	MoveL Offs(p0,126.52000000000001,464.52479999999997, 0), v100, z5, tool0;
	MoveL Offs(p0,127.525,466.325, 0), v100, z5, tool0;
	MoveL Offs(p0,128.584,468.0831999999999, 0), v100, z5, tool0;
	MoveL Offs(p0,129.679,469.7646, 0), v100, z5, tool0;
	MoveL Offs(p0,130.792,471.3344000000001, 0), v100, z5, tool0;
	MoveL Offs(p0,131.90500000000003,472.75780000000003, 0), v100, z5, tool0;
	MoveL Offs(p0,133.0,474.0, 0), v100, z5, tool0;
	MoveL Offs(p0,137.77200000000002,479.7586, 0), v100, z5, tool0;
	MoveL Offs(p0,142.54400000000004,486.68480000000017, 0), v100, z5, tool0;
	MoveL Offs(p0,147.22,494.55420000000004, 0), v100, z5, tool0;
	MoveL Offs(p0,151.704,503.14240000000007, 0), v100, z5, tool0;
	MoveL Offs(p0,155.9,512.225, 0), v100, z5, tool0;
	MoveL Offs(p0,159.712,521.5776, 0), v100, z5, tool0;
	MoveL Offs(p0,163.044,530.9757999999999, 0), v100, z5, tool0;
	MoveL Offs(p0,165.8,540.1952, 0), v100, z5, tool0;
	MoveL Offs(p0,167.884,549.0114000000001, 0), v100, z5, tool0;
	MoveL Offs(p0,169.2,557.2, 0), v100, z5, tool0;
	MoveL Offs(p0,169.67680000000001,561.0432000000002, 0), v100, z5, tool0;
	MoveL Offs(p0,169.9092,562.9168000000001, 0), v100, z5, tool0;
	MoveL Offs(p0,170.1344,564.7136, 0), v100, z5, tool0;
	MoveL Offs(p0,170.35,566.4, 0), v100, z5, tool0;
	MoveL Offs(p0,170.5536,567.9424, 0), v100, z5, tool0;
	MoveL Offs(p0,170.7428,569.3072, 0), v100, z5, tool0;
	MoveL Offs(p0,170.9152,570.4608000000001, 0), v100, z5, tool0;
	MoveL Offs(p0,171.06840000000003,571.3696, 0), v100, z5, tool0;
	MoveL Offs(p0,171.2,572.0, 0), v100, z5, tool0;
	MoveL Offs(p0,171.4976,574.6176, 0), v100, z5, tool0;
	MoveL Offs(p0,171.575,575.425, 0), v100, z5, tool0;
	MoveL Offs(p0,171.6464,576.2624, 0), v100, z5, tool0;
	MoveL Offs(p0,171.7082,577.1142, 0), v100, z5, tool0;
	MoveL Offs(p0,171.75680000000003,577.9648, 0), v100, z5, tool0;
	MoveL Offs(p0,171.78860000000003,578.7986000000001, 0), v100, z5, tool0;
	MoveL Offs(p0,171.8,579.6, 0), v100, z5, tool0;
	MoveL Offs(p0,172.0772,581.6088, 0), v100, z5, tool0;
	MoveL Offs(p0,172.20640000000003,582.1856, 0), v100, z5, tool0;
	MoveL Offs(p0,172.35,582.7, 0), v100, z5, tool0;
	MoveL Offs(p0,172.50560000000002,583.1424, 0), v100, z5, tool0;
	MoveL Offs(p0,172.6708,583.5032, 0), v100, z5, tool0;
	MoveL Offs(p0,172.84320000000002,583.7728000000001, 0), v100, z5, tool0;
	MoveL Offs(p0,173.02040000000002,583.9416, 0), v100, z5, tool0;
	MoveL Offs(p0,173.2,584.0, 0), v100, z5, tool0;
	MoveL Offs(p0,173.70940000000002,581.9156, 0), v100, z5, tool0;
	MoveL Offs(p0,173.7888,580.4032, 0), v100, z5, tool0;
	MoveL Offs(p0,173.825,578.55, 0), v100, z5, tool0;
	MoveL Offs(p0,173.8192,576.3968, 0), v100, z5, tool0;
	MoveL Offs(p0,173.7726,573.9844, 0), v100, z5, tool0;
	MoveL Offs(p0,173.6864,571.3536, 0), v100, z5, tool0;
	MoveL Offs(p0,173.5618,568.5452, 0), v100, z5, tool0;
	MoveL Offs(p0,173.4,565.6, 0), v100, z5, tool0;
	MoveL Offs(p0,173.4,565.6, 0), v100, z5, tool0;
	MoveJ Offs(p0,300.6,571.2, 10), v100, z1, tool0;
	MoveL Offs(p0,301.2482,569.1882, 0), v100, z5, tool0;
	MoveL Offs(p0,301.75360000000006,567.4416000000002, 0), v100, z5, tool0;
	MoveL Offs(p0,302.1174,565.9134000000001, 0), v100, z5, tool0;
	MoveL Offs(p0,302.34080000000006,564.5568000000001, 0), v100, z5, tool0;
	MoveL Offs(p0,302.425,563.325, 0), v100, z5, tool0;
	MoveL Offs(p0,302.37119999999993,562.1712, 0), v100, z5, tool0;
	MoveL Offs(p0,302.18059999999997,561.0486, 0), v100, z5, tool0;
	MoveL Offs(p0,301.85440000000006,559.9104, 0), v100, z5, tool0;
	MoveL Offs(p0,301.3938,558.7098, 0), v100, z5, tool0;
	MoveL Offs(p0,300.8,557.4, 0), v100, z5, tool0;
	MoveL Offs(p0,298.2224,550.942, 0), v100, z5, tool0;
	MoveL Offs(p0,296.3552000000001,542.8880000000001, 0), v100, z5, tool0;
	MoveL Offs(p0,295.1768,533.658, 0), v100, z5, tool0;
	MoveL Offs(p0,294.66560000000004,523.672, 0), v100, z5, tool0;
	MoveL Offs(p0,294.8,513.35, 0), v100, z5, tool0;
	MoveL Offs(p0,295.5584,503.11199999999997, 0), v100, z5, tool0;
	MoveL Offs(p0,296.9192,493.37800000000004, 0), v100, z5, tool0;
	MoveL Offs(p0,298.86080000000004,484.56800000000004, 0), v100, z5, tool0;
	MoveL Offs(p0,301.36160000000007,477.10200000000003, 0), v100, z5, tool0;
	MoveL Offs(p0,304.4,471.4, 0), v100, z5, tool0;
	MoveL Offs(p0,306.18019999999996,468.8188, 0), v100, z5, tool0;
	MoveL Offs(p0,306.66240000000005,468.0496, 0), v100, z5, tool0;
	MoveL Offs(p0,307.075,467.35, 0), v100, z5, tool0;
	MoveL Offs(p0,307.4096,466.7344, 0), v100, z5, tool0;
	MoveL Offs(p0,307.6578,466.21719999999993, 0), v100, z5, tool0;
	MoveL Offs(p0,307.8112,465.81280000000004, 0), v100, z5, tool0;
	MoveL Offs(p0,307.8614,465.53560000000004, 0), v100, z5, tool0;
	MoveL Offs(p0,307.8,465.4, 0), v100, z5, tool0;
	MoveL Offs(p0,305.02880000000005,464.32320000000016, 0), v100, z5, tool0;
	MoveL Offs(p0,302.53319999999997,463.44879999999995, 0), v100, z5, tool0;
	MoveL Offs(p0,299.5984,462.44960000000003, 0), v100, z5, tool0;
	MoveL Offs(p0,296.45,461.4, 0), v100, z5, tool0;
	MoveL Offs(p0,293.3136,460.3744, 0), v100, z5, tool0;
	MoveL Offs(p0,290.4148,459.44719999999995, 0), v100, z5, tool0;
	MoveL Offs(p0,287.97920000000005,458.6928, 0), v100, z5, tool0;
	MoveL Offs(p0,286.2324,458.1856000000001, 0), v100, z5, tool0;
	MoveL Offs(p0,285.4,458.0, 0), v100, z5, tool0;
	MoveL Offs(p0,283.55499999999995,460.51099999999997, 0), v100, z5, tool0;
	MoveL Offs(p0,282.80800000000005,462.32000000000005, 0), v100, z5, tool0;
	MoveL Offs(p0,282.025,464.525, 0), v100, z5, tool0;
	MoveL Offs(p0,281.224,467.072, 0), v100, z5, tool0;
	MoveL Offs(p0,280.423,469.90700000000004, 0), v100, z5, tool0;
	MoveL Offs(p0,279.64000000000004,472.976, 0), v100, z5, tool0;
	MoveL Offs(p0,278.89300000000003,476.225, 0), v100, z5, tool0;
	MoveL Offs(p0,278.2,479.6, 0), v100, z5, tool0;
	MoveL Offs(p0,276.93420000000003,487.9902000000001, 0), v100, z5, tool0;
	MoveL Offs(p0,276.2336000000001,497.66560000000015, 0), v100, z5, tool0;
	MoveL Offs(p0,276.0634,508.2434, 0), v100, z5, tool0;
	MoveL Offs(p0,276.38880000000006,519.3408000000001, 0), v100, z5, tool0;
	MoveL Offs(p0,277.175,530.575, 0), v100, z5, tool0;
	MoveL Offs(p0,278.3872,541.5631999999999, 0), v100, z5, tool0;
	MoveL Offs(p0,279.9906,551.9226, 0), v100, z5, tool0;
	MoveL Offs(p0,281.9504,561.2704, 0), v100, z5, tool0;
	MoveL Offs(p0,284.2318,569.2238, 0), v100, z5, tool0;
	MoveL Offs(p0,286.8,575.4, 0), v100, z5, tool0;
	MoveL Offs(p0,288.153,577.6692, 0), v100, z5, tool0;
	MoveL Offs(p0,289.56000000000006,579.3216000000002, 0), v100, z5, tool0;
	MoveL Offs(p0,291.003,580.3644, 0), v100, z5, tool0;
	MoveL Offs(p0,292.46400000000006,580.8048, 0), v100, z5, tool0;
	MoveL Offs(p0,293.925,580.65, 0), v100, z5, tool0;
	MoveL Offs(p0,295.368,579.9071999999999, 0), v100, z5, tool0;
	MoveL Offs(p0,296.775,578.5836, 0), v100, z5, tool0;
	MoveL Offs(p0,298.12800000000004,576.6864, 0), v100, z5, tool0;
	MoveL Offs(p0,299.409,574.2228000000001, 0), v100, z5, tool0;
	MoveL Offs(p0,300.6,571.2, 0), v100, z5, tool0;
	MoveL Offs(p0,300.6,571.2, 0), v100, z5, tool0;
	MoveJ Offs(p0,313.0,572.2, 10), v100, z1, tool0;
	MoveL Offs(p0,312.6486000000001,570.0876000000001, 0), v100, z5, tool0;
	MoveL Offs(p0,312.56480000000005,568.0448000000001, 0), v100, z5, tool0;
	MoveL Offs(p0,312.76419999999996,566.0332, 0), v100, z5, tool0;
	MoveL Offs(p0,313.2624,564.0143999999999, 0), v100, z5, tool0;
	MoveL Offs(p0,314.075,561.95, 0), v100, z5, tool0;
	MoveL Offs(p0,315.2176,559.8016, 0), v100, z5, tool0;
	MoveL Offs(p0,316.7058,557.5308, 0), v100, z5, tool0;
	MoveL Offs(p0,318.55520000000007,555.0992, 0), v100, z5, tool0;
	MoveL Offs(p0,320.7814,552.4684, 0), v100, z5, tool0;
	MoveL Offs(p0,323.4,549.6, 0), v100, z5, tool0;
	MoveL Offs(p0,325.2538,547.5742000000001, 0), v100, z5, tool0;
	MoveL Offs(p0,326.7344000000001,545.7056000000002, 0), v100, z5, tool0;
	MoveL Offs(p0,327.84059999999994,544.0074000000001, 0), v100, z5, tool0;
	MoveL Offs(p0,328.5712,542.4928, 0), v100, z5, tool0;
	MoveL Offs(p0,328.925,541.175, 0), v100, z5, tool0;
	MoveL Offs(p0,328.9008,540.0672, 0), v100, z5, tool0;
	MoveL Offs(p0,328.4974,539.1826, 0), v100, z5, tool0;
	MoveL Offs(p0,327.71360000000004,538.5344000000001, 0), v100, z5, tool0;
	MoveL Offs(p0,326.54820000000007,538.1358, 0), v100, z5, tool0;
	MoveL Offs(p0,325.0,538.0, 0), v100, z5, tool0;
	MoveL Offs(p0,321.8720000000001,541.2496000000001, 0), v100, z5, tool0;
	MoveL Offs(p0,319.573,544.8093999999999, 0), v100, z5, tool0;
	MoveL Offs(p0,317.016,549.2128, 0), v100, z5, tool0;
	MoveL Offs(p0,314.375,554.125, 0), v100, z5, tool0;
	MoveL Offs(p0,311.824,559.2112, 0), v100, z5, tool0;
	MoveL Offs(p0,309.537,564.1366, 0), v100, z5, tool0;
	MoveL Offs(p0,307.688,568.5664, 0), v100, z5, tool0;
	MoveL Offs(p0,306.451,572.1658, 0), v100, z5, tool0;
	MoveL Offs(p0,306.0,574.6, 0), v100, z5, tool0;
	MoveL Offs(p0,306.7296,576.7472, 0), v100, z5, tool0;
	MoveL Offs(p0,307.125,577.125, 0), v100, z5, tool0;
	MoveL Offs(p0,307.59839999999997,577.4368, 0), v100, z5, tool0;
	MoveL Offs(p0,308.1462,577.6814, 0), v100, z5, tool0;
	MoveL Offs(p0,308.76480000000004,577.8576, 0), v100, z5, tool0;
	MoveL Offs(p0,309.4506,577.9642000000001, 0), v100, z5, tool0;
	MoveL Offs(p0,310.2,578.0, 0), v100, z5, tool0;
	MoveL Offs(p0,312.6192,577.6922, 0), v100, z5, tool0;
	MoveL Offs(p0,313.0864,577.3984, 0), v100, z5, tool0;
	MoveL Offs(p0,313.4,576.975, 0), v100, z5, tool0;
	MoveL Offs(p0,313.56960000000004,576.4015999999999, 0), v100, z5, tool0;
	MoveL Offs(p0,313.60479999999995,575.6578000000001, 0), v100, z5, tool0;
	MoveL Offs(p0,313.5152,574.7232, 0), v100, z5, tool0;
	MoveL Offs(p0,313.3104,573.5774, 0), v100, z5, tool0;
	MoveL Offs(p0,313.0,572.2, 0), v100, z5, tool0;
	MoveL Offs(p0,313.0,572.2, 0), v100, z5, tool0;
	MoveJ Offs(p0,343.8,570.4, 10), v100, z1, tool0;
	MoveL Offs(p0,360.4,567.0, 0), v100, z5, tool0;
	MoveL Offs(p0,348.2,557.2, 0), v100, z5, tool0;
	MoveL Offs(p0,344.5584,554.3928000000002, 0), v100, z5, tool0;
	MoveL Offs(p0,341.5792,552.2144000000001, 0), v100, z5, tool0;
	MoveL Offs(p0,339.1208,550.6696, 0), v100, z5, tool0;
	MoveL Offs(p0,337.0416000000001,549.7632000000001, 0), v100, z5, tool0;
	MoveL Offs(p0,335.2,549.5, 0), v100, z5, tool0;
	MoveL Offs(p0,333.45439999999996,549.8848, 0), v100, z5, tool0;
	MoveL Offs(p0,331.6632,550.9224, 0), v100, z5, tool0;
	MoveL Offs(p0,329.68480000000005,552.6176, 0), v100, z5, tool0;
	MoveL Offs(p0,327.3776,554.9752000000001, 0), v100, z5, tool0;
	MoveL Offs(p0,324.6,558.0, 0), v100, z5, tool0;
	MoveL Offs(p0,322.8896000000001,560.1758000000002, 0), v100, z5, tool0;
	MoveL Offs(p0,321.59680000000014,562.3504000000001, 0), v100, z5, tool0;
	MoveL Offs(p0,320.71919999999994,564.4746, 0), v100, z5, tool0;
	MoveL Offs(p0,320.25440000000003,566.4992, 0), v100, z5, tool0;
	MoveL Offs(p0,320.2,568.375, 0), v100, z5, tool0;
	MoveL Offs(p0,320.55359999999996,570.0527999999999, 0), v100, z5, tool0;
	MoveL Offs(p0,321.3128,571.4834, 0), v100, z5, tool0;
	MoveL Offs(p0,322.47520000000003,572.6176, 0), v100, z5, tool0;
	MoveL Offs(p0,324.0384,573.4062, 0), v100, z5, tool0;
	MoveL Offs(p0,326.0,573.8, 0), v100, z5, tool0;
	MoveL Offs(p0,328.3706,573.4057999999999, 0), v100, z5, tool0;
	MoveL Offs(p0,329.87520000000006,573.1216000000001, 0), v100, z5, tool0;
	MoveL Offs(p0,331.675,572.775, 0), v100, z5, tool0;
	MoveL Offs(p0,333.73279999999994,572.3743999999999, 0), v100, z5, tool0;
	MoveL Offs(p0,336.0114,571.9282000000001, 0), v100, z5, tool0;
	MoveL Offs(p0,338.47360000000003,571.4448, 0), v100, z5, tool0;
	MoveL Offs(p0,341.0822,570.9326, 0), v100, z5, tool0;
	MoveL Offs(p0,343.8,570.4, 0), v100, z5, tool0;
	MoveL Offs(p0,343.8,570.4, 0), v100, z5, tool0;
	MoveJ Offs(p0,145.8,567.6, 10), v100, z1, tool0;
	MoveL Offs(p0,148.6,563.2, 0), v100, z5, tool0;
	MoveL Offs(p0,152.0,567.6, 0), v100, z5, tool0;
	MoveL Offs(p0,154.31040000000002,570.2736000000001, 0), v100, z5, tool0;
	MoveL Offs(p0,155.18959999999998,571.0794, 0), v100, z5, tool0;
	MoveL Offs(p0,155.9392,571.5168000000001, 0), v100, z5, tool0;
	MoveL Offs(p0,156.6,571.575, 0), v100, z5, tool0;
	MoveL Offs(p0,157.2128,571.2432000000001, 0), v100, z5, tool0;
	MoveL Offs(p0,157.8184,570.5106, 0), v100, z5, tool0;
	MoveL Offs(p0,158.4576,569.3664000000001, 0), v100, z5, tool0;
	MoveL Offs(p0,159.1712,567.7998, 0), v100, z5, tool0;
	MoveL Offs(p0,160.0,565.8, 0), v100, z5, tool0;
	MoveL Offs(p0,161.5264,563.019, 0), v100, z5, tool0;
	MoveL Offs(p0,162.06080000000003,562.3120000000001, 0), v100, z5, tool0;
	MoveL Offs(p0,162.6,561.725, 0), v100, z5, tool0;
	MoveL Offs(p0,163.13920000000002,561.2639999999999, 0), v100, z5, tool0;
	MoveL Offs(p0,163.6736,560.9350000000001, 0), v100, z5, tool0;
	MoveL Offs(p0,164.19840000000002,560.744, 0), v100, z5, tool0;
	MoveL Offs(p0,164.70880000000002,560.697, 0), v100, z5, tool0;
	MoveL Offs(p0,165.2,560.8, 0), v100, z5, tool0;
	MoveL Offs(p0,167.2,561.4, 0), v100, z5, tool0;
	MoveL Offs(p0,167.4752,561.4480000000001, 0), v100, z5, tool0;
	MoveL Offs(p0,167.69760000000002,561.472, 0), v100, z5, tool0;
	MoveL Offs(p0,167.86240000000004,561.472, 0), v100, z5, tool0;
	MoveL Offs(p0,167.96480000000003,561.4480000000001, 0), v100, z5, tool0;
	MoveL Offs(p0,168.0,561.4, 0), v100, z5, tool0;
	MoveL Offs(p0,167.65260000000004,558.7860000000001, 0), v100, z5, tool0;
	MoveL Offs(p0,166.68480000000005,554.6480000000001, 0), v100, z5, tool0;
	MoveL Offs(p0,165.20819999999998,549.322, 0), v100, z5, tool0;
	MoveL Offs(p0,163.33440000000002,543.1440000000001, 0), v100, z5, tool0;
	MoveL Offs(p0,161.175,536.45, 0), v100, z5, tool0;
	MoveL Offs(p0,158.8416,529.576, 0), v100, z5, tool0;
	MoveL Offs(p0,156.44580000000002,522.858, 0), v100, z5, tool0;
	MoveL Offs(p0,154.09920000000002,516.632, 0), v100, z5, tool0;
	MoveL Offs(p0,151.9134,511.23400000000004, 0), v100, z5, tool0;
	MoveL Offs(p0,150.0,507.0, 0), v100, z5, tool0;
	MoveL Offs(p0,147.63520000000003,502.4732, 0), v100, z5, tool0;
	MoveL Offs(p0,144.85760000000005,497.68960000000004, 0), v100, z5, tool0;
	MoveL Offs(p0,141.8424,492.8843999999999, 0), v100, z5, tool0;
	MoveL Offs(p0,138.76479999999998,488.29280000000006, 0), v100, z5, tool0;
	MoveL Offs(p0,135.8,484.15, 0), v100, z5, tool0;
	MoveL Offs(p0,133.1232,480.69120000000004, 0), v100, z5, tool0;
	MoveL Offs(p0,130.9096,478.1516, 0), v100, z5, tool0;
	MoveL Offs(p0,129.33440000000002,476.7664000000001, 0), v100, z5, tool0;
	MoveL Offs(p0,128.5728,476.77080000000007, 0), v100, z5, tool0;
	MoveL Offs(p0,128.8,478.4, 0), v100, z5, tool0;
	MoveL Offs(p0,130.18980000000002,484.4408, 0), v100, z5, tool0;
	MoveL Offs(p0,131.35040000000004,492.3824000000001, 0), v100, z5, tool0;
	MoveL Offs(p0,132.2686,501.71360000000004, 0), v100, z5, tool0;
	MoveL Offs(p0,132.93120000000002,511.9232, 0), v100, z5, tool0;
	MoveL Offs(p0,133.325,522.5, 0), v100, z5, tool0;
	MoveL Offs(p0,133.4368,532.9328, 0), v100, z5, tool0;
	MoveL Offs(p0,133.2534,542.7103999999999, 0), v100, z5, tool0;
	MoveL Offs(p0,132.7616,551.3216, 0), v100, z5, tool0;
	MoveL Offs(p0,131.94819999999999,558.2552, 0), v100, z5, tool0;
	MoveL Offs(p0,130.8,563.0, 0), v100, z5, tool0;
	MoveL Offs(p0,130.18880000000001,565.0992, 0), v100, z5, tool0;
	MoveL Offs(p0,130.225,565.375, 0), v100, z5, tool0;
	MoveL Offs(p0,130.3392,565.5487999999999, 0), v100, z5, tool0;
	MoveL Offs(p0,130.5326,565.6193999999999, 0), v100, z5, tool0;
	MoveL Offs(p0,130.8064,565.5856, 0), v100, z5, tool0;
	MoveL Offs(p0,131.16180000000003,565.4462000000001, 0), v100, z5, tool0;
	MoveL Offs(p0,131.6,565.2, 0), v100, z5, tool0;
	MoveL Offs(p0,133.925,565.4, 0), v100, z5, tool0;
	MoveL Offs(p0,134.45120000000003,565.7472, 0), v100, z5, tool0;
	MoveL Offs(p0,134.9726,566.1856, 0), v100, z5, tool0;
	MoveL Offs(p0,135.47840000000002,566.7104, 0), v100, z5, tool0;
	MoveL Offs(p0,135.9578,567.3168, 0), v100, z5, tool0;
	MoveL Offs(p0,136.4,568.0, 0), v100, z5, tool0;
	MoveL Offs(p0,138.28000000000003,570.4736000000001, 0), v100, z5, tool0;
	MoveL Offs(p0,139.19899999999998,571.2274, 0), v100, z5, tool0;
	MoveL Offs(p0,140.11200000000002,571.6608000000001, 0), v100, z5, tool0;
	MoveL Offs(p0,141.025,571.775, 0), v100, z5, tool0;
	MoveL Offs(p0,141.944,571.5712000000001, 0), v100, z5, tool0;
	MoveL Offs(p0,142.875,571.0505999999999, 0), v100, z5, tool0;
	MoveL Offs(p0,143.824,570.2144000000001, 0), v100, z5, tool0;
	MoveL Offs(p0,144.797,569.0638, 0), v100, z5, tool0;
	MoveL Offs(p0,145.8,567.6, 0), v100, z5, tool0;
	MoveL Offs(p0,145.8,567.6, 0), v100, z5, tool0;
	MoveJ Offs(p0,615.0,561.6, 10), v100, z1, tool0;
	MoveL Offs(p0,617.1712000000001,559.1610000000002, 0), v100, z5, tool0;
	MoveL Offs(p0,619.8656000000002,555.5280000000001, 0), v100, z5, tool0;
	MoveL Offs(p0,623.1143999999998,550.6469999999999, 0), v100, z5, tool0;
	MoveL Offs(p0,626.9488,544.464, 0), v100, z5, tool0;
	MoveL Offs(p0,631.4,536.925, 0), v100, z5, tool0;
	MoveL Offs(p0,636.4992,527.976, 0), v100, z5, tool0;
	MoveL Offs(p0,642.2776,517.563, 0), v100, z5, tool0;
	MoveL Offs(p0,648.7664000000001,505.63200000000006, 0), v100, z5, tool0;
	MoveL Offs(p0,655.9968,492.129, 0), v100, z5, tool0;
	MoveL Offs(p0,664.0,477.0, 0), v100, z5, tool0;
	MoveL Offs(p0,667.9796,469.4234, 0), v100, z5, tool0;
	MoveL Offs(p0,671.7168000000003,462.3952000000002, 0), v100, z5, tool0;
	MoveL Offs(p0,675.3292,455.70779999999996, 0), v100, z5, tool0;
	MoveL Offs(p0,678.9344000000001,449.1536000000001, 0), v100, z5, tool0;
	MoveL Offs(p0,682.65,442.525, 0), v100, z5, tool0;
	MoveL Offs(p0,686.5935999999999,435.61440000000005, 0), v100, z5, tool0;
	MoveL Offs(p0,690.8828,428.2142, 0), v100, z5, tool0;
	MoveL Offs(p0,695.6352,420.11679999999996, 0), v100, z5, tool0;
	MoveL Offs(p0,700.9684,411.11460000000005, 0), v100, z5, tool0;
	MoveL Offs(p0,707.0,401.0, 0), v100, z5, tool0;
	MoveL Offs(p0,714.2458000000001,388.87800000000004, 0), v100, z5, tool0;
	MoveL Offs(p0,720.3264000000001,378.5440000000001, 0), v100, z5, tool0;
	MoveL Offs(p0,725.3365999999999,369.8059999999999, 0), v100, z5, tool0;
	MoveL Offs(p0,729.3712,362.472, 0), v100, z5, tool0;
	MoveL Offs(p0,732.525,356.35, 0), v100, z5, tool0;
	MoveL Offs(p0,734.8928,351.248, 0), v100, z5, tool0;
	MoveL Offs(p0,736.5694,346.974, 0), v100, z5, tool0;
	MoveL Offs(p0,737.6496000000001,343.336, 0), v100, z5, tool0;
	MoveL Offs(p0,738.2282,340.142, 0), v100, z5, tool0;
	MoveL Offs(p0,738.4,337.2, 0), v100, z5, tool0;
	MoveL Offs(p0,738.1340000000001,332.6124, 0), v100, z5, tool0;
	MoveL Offs(p0,737.3040000000003,328.29120000000006, 0), v100, z5, tool0;
	MoveL Offs(p0,735.862,324.1788, 0), v100, z5, tool0;
	MoveL Offs(p0,733.7600000000001,320.21760000000006, 0), v100, z5, tool0;
	MoveL Offs(p0,730.95,316.35, 0), v100, z5, tool0;
	MoveL Offs(p0,727.3839999999999,312.5184, 0), v100, z5, tool0;
	MoveL Offs(p0,723.0139999999999,308.6652, 0), v100, z5, tool0;
	MoveL Offs(p0,717.7920000000001,304.73280000000005, 0), v100, z5, tool0;
	MoveL Offs(p0,711.6700000000001,300.66360000000003, 0), v100, z5, tool0;
	MoveL Offs(p0,704.6,296.4, 0), v100, z5, tool0;
	MoveL Offs(p0,694.1098000000001,290.4236, 0), v100, z5, tool0;
	MoveL Offs(p0,683.6304000000002,284.7808000000001, 0), v100, z5, tool0;
	MoveL Offs(p0,673.3285999999999,279.5412, 0), v100, z5, tool0;
	MoveL Offs(p0,663.3711999999999,274.7744, 0), v100, z5, tool0;
	MoveL Offs(p0,653.925,270.55, 0), v100, z5, tool0;
	MoveL Offs(p0,645.1568,266.93760000000003, 0), v100, z5, tool0;
	MoveL Offs(p0,637.2333999999998,264.0068, 0), v100, z5, tool0;
	MoveL Offs(p0,630.3216,261.8272, 0), v100, z5, tool0;
	MoveL Offs(p0,624.5882,260.46840000000003, 0), v100, z5, tool0;
	MoveL Offs(p0,620.2,260.0, 0), v100, z5, tool0;
	MoveL Offs(p0,616.3150000000002,260.21740000000005, 0), v100, z5, tool0;
	MoveL Offs(p0,612.8080000000002,261.04320000000007, 0), v100, z5, tool0;
	MoveL Offs(p0,609.481,262.7378, 0), v100, z5, tool0;
	MoveL Offs(p0,606.136,265.5616, 0), v100, z5, tool0;
	MoveL Offs(p0,602.575,269.775, 0), v100, z5, tool0;
	MoveL Offs(p0,598.6,275.6384, 0), v100, z5, tool0;
	MoveL Offs(p0,594.013,283.41220000000004, 0), v100, z5, tool0;
	MoveL Offs(p0,588.616,293.3568, 0), v100, z5, tool0;
	MoveL Offs(p0,582.211,305.73260000000005, 0), v100, z5, tool0;
	MoveL Offs(p0,574.6,320.8, 0), v100, z5, tool0;
	MoveL Offs(p0,570.4530000000002,329.05840000000006, 0), v100, z5, tool0;
	MoveL Offs(p0,566.336,337.1872000000001, 0), v100, z5, tool0;
	MoveL Offs(p0,562.3149999999999,345.05679999999995, 0), v100, z5, tool0;
	MoveL Offs(p0,558.4560000000001,352.5376, 0), v100, z5, tool0;
	MoveL Offs(p0,554.825,359.5, 0), v100, z5, tool0;
	MoveL Offs(p0,551.488,365.8144, 0), v100, z5, tool0;
	MoveL Offs(p0,548.511,371.35119999999995, 0), v100, z5, tool0;
	MoveL Offs(p0,545.96,375.9808, 0), v100, z5, tool0;
	MoveL Offs(p0,543.9010000000001,379.5736, 0), v100, z5, tool0;
	MoveL Offs(p0,542.4,382.0, 0), v100, z5, tool0;
	MoveL Offs(p0,537.9362000000001,388.80320000000006, 0), v100, z5, tool0;
	MoveL Offs(p0,532.5136000000001,396.63360000000006, 0), v100, z5, tool0;
	MoveL Offs(p0,526.3853999999999,405.1624, 0), v100, z5, tool0;
	MoveL Offs(p0,519.8048000000001,414.06080000000003, 0), v100, z5, tool0;
	MoveL Offs(p0,513.025,423.0, 0), v100, z5, tool0;
	MoveL Offs(p0,506.2991999999999,431.65119999999996, 0), v100, z5, tool0;
	MoveL Offs(p0,499.88059999999996,439.68559999999997, 0), v100, z5, tool0;
	MoveL Offs(p0,494.0224,446.77440000000007, 0), v100, z5, tool0;
	MoveL Offs(p0,488.9778,452.5888000000001, 0), v100, z5, tool0;
	MoveL Offs(p0,485.0,456.8, 0), v100, z5, tool0;
	MoveL Offs(p0,481.7126,460.1758, 0), v100, z5, tool0;
	MoveL Offs(p0,478.90880000000016,463.2624000000002, 0), v100, z5, tool0;
	MoveL Offs(p0,476.5561999999999,466.1185999999999, 0), v100, z5, tool0;
	MoveL Offs(p0,474.6224,468.8032, 0), v100, z5, tool0;
	MoveL Offs(p0,473.075,471.375, 0), v100, z5, tool0;
	MoveL Offs(p0,471.8816,473.89279999999997, 0), v100, z5, tool0;
	MoveL Offs(p0,471.0098,476.41540000000003, 0), v100, z5, tool0;
	MoveL Offs(p0,470.4272000000001,479.00159999999994, 0), v100, z5, tool0;
	MoveL Offs(p0,470.1014000000001,481.7102, 0), v100, z5, tool0;
	MoveL Offs(p0,470.0,484.6, 0), v100, z5, tool0;
	MoveL Offs(p0,470.2696000000001,487.9942, 0), v100, z5, tool0;
	MoveL Offs(p0,470.9808000000001,490.99360000000013, 0), v100, z5, tool0;
	MoveL Offs(p0,472.16720000000004,493.62339999999995, 0), v100, z5, tool0;
	MoveL Offs(p0,473.8624,495.90880000000004, 0), v100, z5, tool0;
	MoveL Offs(p0,476.1,497.875, 0), v100, z5, tool0;
	MoveL Offs(p0,478.91360000000003,499.5472, 0), v100, z5, tool0;
	MoveL Offs(p0,482.33680000000004,500.9506, 0), v100, z5, tool0;
	MoveL Offs(p0,486.4032000000001,502.1104, 0), v100, z5, tool0;
	MoveL Offs(p0,491.14639999999997,503.0518, 0), v100, z5, tool0;
	MoveL Offs(p0,496.6,503.8, 0), v100, z5, tool0;
	MoveL Offs(p0,500.0086,504.24860000000007, 0), v100, z5, tool0;
	MoveL Offs(p0,503.20480000000015,504.7728000000001, 0), v100, z5, tool0;
	MoveL Offs(p0,506.26419999999996,505.4001999999999, 0), v100, z5, tool0;
	MoveL Offs(p0,509.26240000000007,506.1584000000001, 0), v100, z5, tool0;
	MoveL Offs(p0,512.275,507.075, 0), v100, z5, tool0;
	MoveL Offs(p0,515.3776,508.1776, 0), v100, z5, tool0;
	MoveL Offs(p0,518.6458,509.4938, 0), v100, z5, tool0;
	MoveL Offs(p0,522.1552,511.05120000000005, 0), v100, z5, tool0;
	MoveL Offs(p0,525.9814,512.8774000000001, 0), v100, z5, tool0;
	MoveL Offs(p0,530.2,515.0, 0), v100, z5, tool0;
	MoveL Offs(p0,537.9566000000001,519.0342, 0), v100, z5, tool0;
	MoveL Offs(p0,544.9488,522.8896000000002, 0), v100, z5, tool0;
	MoveL Offs(p0,551.2402,526.6154, 0), v100, z5, tool0;
	MoveL Offs(p0,556.8944,530.2607999999999, 0), v100, z5, tool0;
	MoveL Offs(p0,561.975,533.875, 0), v100, z5, tool0;
	MoveL Offs(p0,566.5456,537.5072, 0), v100, z5, tool0;
	MoveL Offs(p0,570.6698,541.2066000000001, 0), v100, z5, tool0;
	MoveL Offs(p0,574.4112000000001,545.0224000000001, 0), v100, z5, tool0;
	MoveL Offs(p0,577.8334000000001,549.0038000000001, 0), v100, z5, tool0;
	MoveL Offs(p0,581.0,553.2, 0), v100, z5, tool0;
	MoveL Offs(p0,583.6990000000001,556.9082000000001, 0), v100, z5, tool0;
	MoveL Offs(p0,585.9840000000002,559.9216000000001, 0), v100, z5, tool0;
	MoveL Offs(p0,587.957,562.3134, 0), v100, z5, tool0;
	MoveL Offs(p0,589.72,564.1568, 0), v100, z5, tool0;
	MoveL Offs(p0,591.375,565.525, 0), v100, z5, tool0;
	MoveL Offs(p0,593.024,566.4912, 0), v100, z5, tool0;
	MoveL Offs(p0,594.769,567.1286, 0), v100, z5, tool0;
	MoveL Offs(p0,596.7120000000001,567.5104000000001, 0), v100, z5, tool0;
	MoveL Offs(p0,598.955,567.7098, 0), v100, z5, tool0;
	MoveL Offs(p0,601.6,567.8, 0), v100, z5, tool0;
	MoveL Offs(p0,604.2800000000002,567.6736000000001, 0), v100, z5, tool0;
	MoveL Offs(p0,605.578,567.4184, 0), v100, z5, tool0;
	MoveL Offs(p0,606.864,567.0288, 0), v100, z5, tool0;
	MoveL Offs(p0,608.15,566.5, 0), v100, z5, tool0;
	MoveL Offs(p0,609.448,565.8272, 0), v100, z5, tool0;
	MoveL Offs(p0,610.77,565.0056, 0), v100, z5, tool0;
	MoveL Offs(p0,612.128,564.0304, 0), v100, z5, tool0;
	MoveL Offs(p0,613.534,562.8968, 0), v100, z5, tool0;
	MoveL Offs(p0,615.0,561.6, 0), v100, z5, tool0;
	MoveL Offs(p0,615.0,561.6, 0), v100, z5, tool0;
	MoveJ Offs(p0,378.6,562.8, 10), v100, z1, tool0;
	MoveL Offs(p0,381.08939999999996,562.0818, 0), v100, z5, tool0;
	MoveL Offs(p0,381.7968,561.7855999999999, 0), v100, z5, tool0;
	MoveL Offs(p0,382.425,561.475, 0), v100, z5, tool0;
	MoveL Offs(p0,382.96320000000003,561.1584, 0), v100, z5, tool0;
	MoveL Offs(p0,383.4006,560.8442, 0), v100, z5, tool0;
	MoveL Offs(p0,383.7264,560.5408000000001, 0), v100, z5, tool0;
	MoveL Offs(p0,383.92980000000006,560.2566, 0), v100, z5, tool0;
	MoveL Offs(p0,384.0,560.0, 0), v100, z5, tool0;
	MoveL Offs(p0,382.35840000000013,556.3552000000002, 0), v100, z5, tool0;
	MoveL Offs(p0,380.45759999999996,553.6748, 0), v100, z5, tool0;
	MoveL Offs(p0,377.9712,550.5696, 0), v100, z5, tool0;
	MoveL Offs(p0,375.0,547.15, 0), v100, z5, tool0;
	MoveL Offs(p0,371.6448,543.5264, 0), v100, z5, tool0;
	MoveL Offs(p0,368.0064,539.8092, 0), v100, z5, tool0;
	MoveL Offs(p0,364.1856000000001,536.1088000000001, 0), v100, z5, tool0;
	MoveL Offs(p0,360.2832,532.5355999999999, 0), v100, z5, tool0;
	MoveL Offs(p0,356.4,529.2, 0), v100, z5, tool0;
	MoveL Offs(p0,352.17820000000006,525.844, 0), v100, z5, tool0;
	MoveL Offs(p0,348.6656000000001,523.2080000000001, 0), v100, z5, tool0;
	MoveL Offs(p0,345.7314,521.28, 0), v100, z5, tool0;
	MoveL Offs(p0,343.24480000000005,520.048, 0), v100, z5, tool0;
	MoveL Offs(p0,341.075,519.5, 0), v100, z5, tool0;
	MoveL Offs(p0,339.09119999999996,519.624, 0), v100, z5, tool0;
	MoveL Offs(p0,337.16259999999994,520.408, 0), v100, z5, tool0;
	MoveL Offs(p0,335.15840000000003,521.84, 0), v100, z5, tool0;
	MoveL Offs(p0,332.94780000000003,523.908, 0), v100, z5, tool0;
	MoveL Offs(p0,330.4,526.6, 0), v100, z5, tool0;
	MoveL Offs(p0,325.8,531.4, 0), v100, z5, tool0;
	MoveL Offs(p0,344.8,546.8, 0), v100, z5, tool0;
	MoveL Offs(p0,347.8766,549.296, 0), v100, z5, tool0;
	MoveL Offs(p0,350.8368000000001,551.7200000000001, 0), v100, z5, tool0;
	MoveL Offs(p0,353.63620000000003,554.036, 0), v100, z5, tool0;
	MoveL Offs(p0,356.23040000000003,556.208, 0), v100, z5, tool0;
	MoveL Offs(p0,358.575,558.2, 0), v100, z5, tool0;
	MoveL Offs(p0,360.6256,559.976, 0), v100, z5, tool0;
	MoveL Offs(p0,362.33779999999996,561.5, 0), v100, z5, tool0;
	MoveL Offs(p0,363.66720000000004,562.7360000000001, 0), v100, z5, tool0;
	MoveL Offs(p0,364.56940000000003,563.648, 0), v100, z5, tool0;
	MoveL Offs(p0,365.0,564.2, 0), v100, z5, tool0;
	MoveL Offs(p0,367.43359999999996,565.3951999999999, 0), v100, z5, tool0;
	MoveL Offs(p0,367.9638,565.4376, 0), v100, z5, tool0;
	MoveL Offs(p0,368.5072,565.4224, 0), v100, z5, tool0;
	MoveL Offs(p0,369.0554,565.3448000000001, 0), v100, z5, tool0;
	MoveL Offs(p0,369.6,565.2, 0), v100, z5, tool0;
	MoveL Offs(p0,371.8212,564.5681999999999, 0), v100, z5, tool0;
	MoveL Offs(p0,372.71040000000005,564.3264, 0), v100, z5, tool0;
	MoveL Offs(p0,373.65,564.075, 0), v100, z5, tool0;
	MoveL Offs(p0,374.62559999999996,563.8176, 0), v100, z5, tool0;
	MoveL Offs(p0,375.6228,563.5577999999999, 0), v100, z5, tool0;
	MoveL Offs(p0,376.6272,563.2992, 0), v100, z5, tool0;
	MoveL Offs(p0,377.6244,563.0454000000001, 0), v100, z5, tool0;
	MoveL Offs(p0,378.6,562.8, 0), v100, z5, tool0;
	MoveL Offs(p0,378.6,562.8, 0), v100, z5, tool0;
	MoveJ Offs(p0,579.4,563.2, 10), v100, z1, tool0;
	MoveL Offs(p0,579.1984000000001,560.5936000000002, 0), v100, z5, tool0;
	MoveL Offs(p0,578.1076,558.4354000000001, 0), v100, z5, tool0;
	MoveL Offs(p0,576.4912,555.8848, 0), v100, z5, tool0;
	MoveL Offs(p0,574.45,553.075, 0), v100, z5, tool0;
	MoveL Offs(p0,572.0848,550.1392, 0), v100, z5, tool0;
	MoveL Offs(p0,569.4964,547.2106, 0), v100, z5, tool0;
	MoveL Offs(p0,566.7856,544.4224, 0), v100, z5, tool0;
	MoveL Offs(p0,564.0532000000001,541.9078, 0), v100, z5, tool0;
	MoveL Offs(p0,561.4,539.8, 0), v100, z5, tool0;
	MoveL Offs(p0,557.7360000000001,537.3040000000002, 0), v100, z5, tool0;
	MoveL Offs(p0,555.3159999999999,535.7679999999999, 0), v100, z5, tool0;
	MoveL Offs(p0,552.5840000000001,534.088, 0), v100, z5, tool0;
	MoveL Offs(p0,549.6,532.3, 0), v100, z5, tool0;
	MoveL Offs(p0,546.424,530.4399999999999, 0), v100, z5, tool0;
	MoveL Offs(p0,543.116,528.544, 0), v100, z5, tool0;
	MoveL Offs(p0,539.7360000000001,526.648, 0), v100, z5, tool0;
	MoveL Offs(p0,536.344,524.788, 0), v100, z5, tool0;
	MoveL Offs(p0,533.0,523.0, 0), v100, z5, tool0;
	MoveL Offs(p0,528.5562000000001,520.6444, 0), v100, z5, tool0;
	MoveL Offs(p0,524.5456000000001,518.6032000000002, 0), v100, z5, tool0;
	MoveL Offs(p0,520.9094,516.8548, 0), v100, z5, tool0;
	MoveL Offs(p0,517.5888,515.3776, 0), v100, z5, tool0;
	MoveL Offs(p0,514.525,514.15, 0), v100, z5, tool0;
	MoveL Offs(p0,511.65919999999994,513.1504, 0), v100, z5, tool0;
	MoveL Offs(p0,508.9326,512.3572, 0), v100, z5, tool0;
	MoveL Offs(p0,506.28640000000007,511.7488, 0), v100, z5, tool0;
	MoveL Offs(p0,503.6618,511.3036, 0), v100, z5, tool0;
	MoveL Offs(p0,501.0,511.0, 0), v100, z5, tool0;
	MoveL Offs(p0,498.98420000000016,510.7430000000001, 0), v100, z5, tool0;
	MoveL Offs(p0,496.92160000000024,510.45600000000013, 0), v100, z5, tool0;
	MoveL Offs(p0,494.84939999999995,510.145, 0), v100, z5, tool0;
	MoveL Offs(p0,492.80480000000006,509.8160000000001, 0), v100, z5, tool0;
	MoveL Offs(p0,490.825,509.475, 0), v100, z5, tool0;
	MoveL Offs(p0,488.94719999999995,509.128, 0), v100, z5, tool0;
	MoveL Offs(p0,487.20859999999993,508.78099999999995, 0), v100, z5, tool0;
	MoveL Offs(p0,485.64639999999997,508.44000000000005, 0), v100, z5, tool0;
	MoveL Offs(p0,484.2978,508.11100000000005, 0), v100, z5, tool0;
	MoveL Offs(p0,483.2,507.8, 0), v100, z5, tool0;
	MoveL Offs(p0,477.6,506.0, 0), v100, z5, tool0;
	MoveL Offs(p0,479.0,513.4, 0), v100, z5, tool0;
	MoveL Offs(p0,479.55459999999994,515.9362000000001, 0), v100, z5, tool0;
	MoveL Offs(p0,480.2448000000001,518.4736000000001, 0), v100, z5, tool0;
	MoveL Offs(p0,481.05019999999996,520.9653999999999, 0), v100, z5, tool0;
	MoveL Offs(p0,481.95040000000006,523.3648000000001, 0), v100, z5, tool0;
	MoveL Offs(p0,482.925,525.625, 0), v100, z5, tool0;
	MoveL Offs(p0,483.9536,527.6992, 0), v100, z5, tool0;
	MoveL Offs(p0,485.01579999999996,529.5406, 0), v100, z5, tool0;
	MoveL Offs(p0,486.0912,531.1024000000001, 0), v100, z5, tool0;
	MoveL Offs(p0,487.1594,532.3378, 0), v100, z5, tool0;
	MoveL Offs(p0,488.2,533.2, 0), v100, z5, tool0;
	MoveL Offs(p0,491.0458,533.8066000000001, 0), v100, z5, tool0;
	MoveL Offs(p0,492.67359999999996,533.9552, 0), v100, z5, tool0;
	MoveL Offs(p0,494.575,534.075, 0), v100, z5, tool0;
	MoveL Offs(p0,496.71039999999994,534.1648, 0), v100, z5, tool0;
	MoveL Offs(p0,499.0402,534.2234000000001, 0), v100, z5, tool0;
	MoveL Offs(p0,501.5248,534.2496000000001, 0), v100, z5, tool0;
	MoveL Offs(p0,504.1246,534.2422, 0), v100, z5, tool0;
	MoveL Offs(p0,506.8,534.2, 0), v100, z5, tool0;
	MoveL Offs(p0,512.3294000000001,534.1712000000001, 0), v100, z5, tool0;
	MoveL Offs(p0,517.0032000000001,534.3776000000001, 0), v100, z5, tool0;
	MoveL Offs(p0,520.9498,534.8983999999999, 0), v100, z5, tool0;
	MoveL Offs(p0,524.2976,535.8128, 0), v100, z5, tool0;
	MoveL Offs(p0,527.175,537.2, 0), v100, z5, tool0;
	MoveL Offs(p0,529.7104,539.1392, 0), v100, z5, tool0;
	MoveL Offs(p0,532.0322,541.7096, 0), v100, z5, tool0;
	MoveL Offs(p0,534.2688,544.9904, 0), v100, z5, tool0;
	MoveL Offs(p0,536.5486,549.0608, 0), v100, z5, tool0;
	MoveL Offs(p0,539.0,554.0, 0), v100, z5, tool0;
	MoveL Offs(p0,545.0,566.6, 0), v100, z5, tool0;
	MoveL Offs(p0,561.6,565.4, 0), v100, z5, tool0;
	MoveL Offs(p0,564.3178,565.2088, 0), v100, z5, tool0;
	MoveL Offs(p0,566.9264000000001,564.9984000000002, 0), v100, z5, tool0;
	MoveL Offs(p0,569.3886,564.7736, 0), v100, z5, tool0;
	MoveL Offs(p0,571.6672000000001,564.5391999999999, 0), v100, z5, tool0;
	MoveL Offs(p0,573.725,564.3, 0), v100, z5, tool0;
	MoveL Offs(p0,575.5248,564.0608, 0), v100, z5, tool0;
	MoveL Offs(p0,577.0294,563.8264, 0), v100, z5, tool0;
	MoveL Offs(p0,578.2016000000001,563.6016000000001, 0), v100, z5, tool0;
	MoveL Offs(p0,579.0042000000001,563.3912, 0), v100, z5, tool0;
	MoveL Offs(p0,579.4,563.2, 0), v100, z5, tool0;
	MoveL Offs(p0,579.4,563.2, 0), v100, z5, tool0;
	MoveJ Offs(p0,409.0,556.4, 10), v100, z1, tool0;
	MoveL Offs(p0,412.6224000000001,555.4976, 0), v100, z5, tool0;
	MoveL Offs(p0,414.0795999999999,554.9294, 0), v100, z5, tool0;
	MoveL Offs(p0,415.37120000000004,554.2208, 0), v100, z5, tool0;
	MoveL Offs(p0,416.55,553.325, 0), v100, z5, tool0;
	MoveL Offs(p0,417.66880000000003,552.1952, 0), v100, z5, tool0;
	MoveL Offs(p0,418.7804,550.7846, 0), v100, z5, tool0;
	MoveL Offs(p0,419.93760000000003,549.0464, 0), v100, z5, tool0;
	MoveL Offs(p0,421.1932,546.9338, 0), v100, z5, tool0;
	MoveL Offs(p0,422.6,544.4, 0), v100, z5, tool0;
	MoveL Offs(p0,426.5228,537.9682, 0), v100, z5, tool0;
	MoveL Offs(p0,430.99040000000014,531.9456000000001, 0), v100, z5, tool0;
	MoveL Offs(p0,435.85159999999996,526.4413999999999, 0), v100, z5, tool0;
	MoveL Offs(p0,440.95520000000005,521.5648, 0), v100, z5, tool0;
	MoveL Offs(p0,446.15,517.425, 0), v100, z5, tool0;
	MoveL Offs(p0,451.2848,514.1312, 0), v100, z5, tool0;
	MoveL Offs(p0,456.2084,511.79259999999994, 0), v100, z5, tool0;
	MoveL Offs(p0,460.76959999999997,510.5184000000001, 0), v100, z5, tool0;
	MoveL Offs(p0,464.81720000000007,510.4178, 0), v100, z5, tool0;
	MoveL Offs(p0,468.2,511.6, 0), v100, z5, tool0;
	MoveL Offs(p0,470.80000000000007,513.1024000000001, 0), v100, z5, tool0;
	MoveL Offs(p0,471.746,513.5296, 0), v100, z5, tool0;
	MoveL Offs(p0,472.488,513.7312000000001, 0), v100, z5, tool0;
	MoveL Offs(p0,473.05,513.7, 0), v100, z5, tool0;
	MoveL Offs(p0,473.45599999999996,513.4288, 0), v100, z5, tool0;
	MoveL Offs(p0,473.73,512.9104, 0), v100, z5, tool0;
	MoveL Offs(p0,473.8960000000001,512.1376, 0), v100, z5, tool0;
	MoveL Offs(p0,473.97800000000007,511.1032, 0), v100, z5, tool0;
	MoveL Offs(p0,474.0,509.8, 0), v100, z5, tool0;
	MoveL Offs(p0,473.4492,507.12340000000006, 0), v100, z5, tool0;
	MoveL Offs(p0,473.0464,505.98879999999997, 0), v100, z5, tool0;
	MoveL Offs(p0,472.55,504.775, 0), v100, z5, tool0;
	MoveL Offs(p0,471.9696,503.5072, 0), v100, z5, tool0;
	MoveL Offs(p0,471.31479999999993,502.2106, 0), v100, z5, tool0;
	MoveL Offs(p0,470.59520000000003,500.91040000000004, 0), v100, z5, tool0;
	MoveL Offs(p0,469.82039999999995,499.6318, 0), v100, z5, tool0;
	MoveL Offs(p0,469.0,498.4, 0), v100, z5, tool0;
	MoveL Offs(p0,467.5122,495.93680000000006, 0), v100, z5, tool0;
	MoveL Offs(p0,466.2896000000002,493.3584000000002, 0), v100, z5, tool0;
	MoveL Offs(p0,465.3334,490.6816, 0), v100, z5, tool0;
	MoveL Offs(p0,464.64480000000003,487.92320000000007, 0), v100, z5, tool0;
	MoveL Offs(p0,464.225,485.1, 0), v100, z5, tool0;
	MoveL Offs(p0,464.07519999999994,482.22880000000004, 0), v100, z5, tool0;
	MoveL Offs(p0,464.19660000000005,479.3263999999999, 0), v100, z5, tool0;
	MoveL Offs(p0,464.59040000000005,476.40960000000007, 0), v100, z5, tool0;
	MoveL Offs(p0,465.25780000000003,473.4952, 0), v100, z5, tool0;
	MoveL Offs(p0,466.2,470.6, 0), v100, z5, tool0;
	MoveL Offs(p0,467.5408000000001,468.0928000000002, 0), v100, z5, tool0;
	MoveL Offs(p0,468.70919999999995,466.3772, 0), v100, z5, tool0;
	MoveL Offs(p0,470.1584000000001,464.4144, 0), v100, z5, tool0;
	MoveL Offs(p0,471.85,462.25, 0), v100, z5, tool0;
	MoveL Offs(p0,473.7456,459.92960000000005, 0), v100, z5, tool0;
	MoveL Offs(p0,475.8068,457.49879999999996, 0), v100, z5, tool0;
	MoveL Offs(p0,477.9952000000001,455.0032, 0), v100, z5, tool0;
	MoveL Offs(p0,480.2724,452.4884, 0), v100, z5, tool0;
	MoveL Offs(p0,482.6,450.0, 0), v100, z5, tool0;
	MoveL Offs(p0,486.43520000000007,445.99760000000003, 0), v100, z5, tool0;
	MoveL Offs(p0,490.1216000000001,442.0528000000001, 0), v100, z5, tool0;
	MoveL Offs(p0,493.6304,438.1991999999999, 0), v100, z5, tool0;
	MoveL Offs(p0,496.93280000000016,434.4704, 0), v100, z5, tool0;
	MoveL Offs(p0,500.0,430.9, 0), v100, z5, tool0;
	MoveL Offs(p0,502.8032,427.52160000000003, 0), v100, z5, tool0;
	MoveL Offs(p0,505.31360000000006,424.3688, 0), v100, z5, tool0;
	MoveL Offs(p0,507.50240000000014,421.47520000000003, 0), v100, z5, tool0;
	MoveL Offs(p0,509.34080000000006,418.87440000000004, 0), v100, z5, tool0;
	MoveL Offs(p0,510.8,416.6, 0), v100, z5, tool0;
	MoveL Offs(p0,507.1264,416.8848, 0), v100, z5, tool0;
	MoveL Offs(p0,507.0272,417.22440000000006, 0), v100, z5, tool0;
	MoveL Offs(p0,507.00480000000005,417.5616, 0), v100, z5, tool0;
	MoveL Offs(p0,507.0616,417.88919999999996, 0), v100, z5, tool0;
	MoveL Offs(p0,507.2,418.2, 0), v100, z5, tool0;
	MoveL Offs(p0,504.8348,419.97659999999996, 0), v100, z5, tool0;
	MoveL Offs(p0,504.2,420.0, 0), v100, z5, tool0;
	MoveL Offs(p0,501.6848,420.4416000000001, 0), v100, z5, tool0;
	MoveL Offs(p0,501.2,420.675, 0), v100, z5, tool0;
	MoveL Offs(p0,500.7871999999999,420.95040000000006, 0), v100, z5, tool0;
	MoveL Offs(p0,500.4536,421.26419999999996, 0), v100, z5, tool0;
	MoveL Offs(p0,500.20640000000003,421.61280000000005, 0), v100, z5, tool0;
	MoveL Offs(p0,500.05280000000005,421.99260000000004, 0), v100, z5, tool0;
	MoveL Offs(p0,500.0,422.4, 0), v100, z5, tool0;
	MoveL Offs(p0,496.6528,423.3008, 0), v100, z5, tool0;
	MoveL Offs(p0,495.75,423.45, 0), v100, z5, tool0;
	MoveL Offs(p0,494.7392,423.65920000000006, 0), v100, z5, tool0;
	MoveL Offs(p0,493.6396,423.9236000000001, 0), v100, z5, tool0;
	MoveL Offs(p0,492.47040000000004,424.2384, 0), v100, z5, tool0;
	MoveL Offs(p0,491.25079999999997,424.59880000000004, 0), v100, z5, tool0;
	MoveL Offs(p0,490.0,425.0, 0), v100, z5, tool0;
	MoveL Offs(p0,487.3510000000001,425.79620000000006, 0), v100, z5, tool0;
	MoveL Offs(p0,484.2880000000002,426.49760000000015, 0), v100, z5, tool0;
	MoveL Offs(p0,480.937,427.09340000000003, 0), v100, z5, tool0;
	MoveL Offs(p0,477.424,427.57280000000003, 0), v100, z5, tool0;
	MoveL Offs(p0,473.875,427.925, 0), v100, z5, tool0;
	MoveL Offs(p0,470.416,428.13919999999996, 0), v100, z5, tool0;
	MoveL Offs(p0,467.17299999999994,428.2046, 0), v100, z5, tool0;
	MoveL Offs(p0,464.2720000000001,428.1104, 0), v100, z5, tool0;
	MoveL Offs(p0,461.83900000000006,427.84580000000005, 0), v100, z5, tool0;
	MoveL Offs(p0,460.0,427.4, 0), v100, z5, tool0;
	MoveL Offs(p0,452.0402000000001,424.7006, 0), v100, z5, tool0;
	MoveL Offs(p0,445.5456000000002,422.60480000000007, 0), v100, z5, tool0;
	MoveL Offs(p0,440.3134,421.11619999999994, 0), v100, z5, tool0;
	MoveL Offs(p0,436.1408,420.2384, 0), v100, z5, tool0;
	MoveL Offs(p0,432.825,419.975, 0), v100, z5, tool0;
	MoveL Offs(p0,430.16319999999996,420.3296, 0), v100, z5, tool0;
	MoveL Offs(p0,427.95259999999996,421.3058, 0), v100, z5, tool0;
	MoveL Offs(p0,425.9904,422.9072, 0), v100, z5, tool0;
	MoveL Offs(p0,424.0738,425.13739999999996, 0), v100, z5, tool0;
	MoveL Offs(p0,422.0,428.0, 0), v100, z5, tool0;
	MoveL Offs(p0,417.8,434.0, 0), v100, z5, tool0;
	MoveL Offs(p0,424.8,440.2, 0), v100, z5, tool0;
	MoveL Offs(p0,427.1826000000001,442.38520000000005, 0), v100, z5, tool0;
	MoveL Offs(p0,429.0528000000001,444.4336000000001, 0), v100, z5, tool0;
	MoveL Offs(p0,430.41420000000005,446.42440000000005, 0), v100, z5, tool0;
	MoveL Offs(p0,431.27040000000005,448.43680000000006, 0), v100, z5, tool0;
	MoveL Offs(p0,431.625,450.55, 0), v100, z5, tool0;
	MoveL Offs(p0,431.48159999999996,452.84319999999997, 0), v100, z5, tool0;
	MoveL Offs(p0,430.8438,455.3956, 0), v100, z5, tool0;
	MoveL Offs(p0,429.7152,458.28639999999996, 0), v100, z5, tool0;
	MoveL Offs(p0,428.09940000000006,461.5948, 0), v100, z5, tool0;
	MoveL Offs(p0,426.0,465.4, 0), v100, z5, tool0;
	MoveL Offs(p0,422.3746,470.98480000000006, 0), v100, z5, tool0;
	MoveL Offs(p0,418.3808000000001,475.63840000000016, 0), v100, z5, tool0;
	MoveL Offs(p0,413.9022,479.3896, 0), v100, z5, tool0;
	MoveL Offs(p0,408.8224,482.26720000000006, 0), v100, z5, tool0;
	MoveL Offs(p0,403.025,484.3, 0), v100, z5, tool0;
	MoveL Offs(p0,396.3936,485.5168, 0), v100, z5, tool0;
	MoveL Offs(p0,388.81180000000006,485.9464, 0), v100, z5, tool0;
	MoveL Offs(p0,380.1632000000001,485.61760000000004, 0), v100, z5, tool0;
	MoveL Offs(p0,370.33140000000003,484.55920000000003, 0), v100, z5, tool0;
	MoveL Offs(p0,359.2,482.8, 0), v100, z5, tool0;
	MoveL Offs(p0,341.4,479.8, 0), v100, z5, tool0;
	MoveL Offs(p0,335.8,485.4, 0), v100, z5, tool0;
	MoveL Offs(p0,333.12180000000006,488.2960000000001, 0), v100, z5, tool0;
	MoveL Offs(p0,331.1024000000001,490.8080000000001, 0), v100, z5, tool0;
	MoveL Offs(p0,329.7646,493.032, 0), v100, z5, tool0;
	MoveL Offs(p0,329.13120000000004,495.064, 0), v100, z5, tool0;
	MoveL Offs(p0,329.225,497.0, 0), v100, z5, tool0;
	MoveL Offs(p0,330.0688,498.93600000000004, 0), v100, z5, tool0;
	MoveL Offs(p0,331.6854,500.968, 0), v100, z5, tool0;
	MoveL Offs(p0,334.0976,503.192, 0), v100, z5, tool0;
	MoveL Offs(p0,337.32820000000004,505.704, 0), v100, z5, tool0;
	MoveL Offs(p0,341.4,508.6, 0), v100, z5, tool0;
	MoveL Offs(p0,346.22159999999997,512.0968, 0), v100, z5, tool0;
	MoveL Offs(p0,351.6528000000001,516.4384000000001, 0), v100, z5, tool0;
	MoveL Offs(p0,357.46320000000003,521.4015999999999, 0), v100, z5, tool0;
	MoveL Offs(p0,363.42240000000004,526.7632000000001, 0), v100, z5, tool0;
	MoveL Offs(p0,369.3,532.3, 0), v100, z5, tool0;
	MoveL Offs(p0,374.8656,537.7887999999999, 0), v100, z5, tool0;
	MoveL Offs(p0,379.8888,543.0064, 0), v100, z5, tool0;
	MoveL Offs(p0,384.1392000000001,547.7296, 0), v100, z5, tool0;
	MoveL Offs(p0,387.38640000000004,551.7352000000001, 0), v100, z5, tool0;
	MoveL Offs(p0,389.4,554.8, 0), v100, z5, tool0;
	MoveL Offs(p0,390.59040000000016,556.8496000000002, 0), v100, z5, tool0;
	MoveL Offs(p0,391.1945999999999,557.6224, 0), v100, z5, tool0;
	MoveL Offs(p0,391.8192,558.2368, 0), v100, z5, tool0;
	MoveL Offs(p0,392.475,558.7, 0), v100, z5, tool0;
	MoveL Offs(p0,393.1728,559.0192, 0), v100, z5, tool0;
	MoveL Offs(p0,393.9234,559.2016, 0), v100, z5, tool0;
	MoveL Offs(p0,394.73760000000004,559.2544, 0), v100, z5, tool0;
	MoveL Offs(p0,395.62620000000004,559.1848, 0), v100, z5, tool0;
	MoveL Offs(p0,396.6,559.0, 0), v100, z5, tool0;
	MoveL Offs(p0,399.50519999999995,558.3249999999999, 0), v100, z5, tool0;
	MoveL Offs(p0,400.73440000000005,558.056, 0), v100, z5, tool0;
	MoveL Offs(p0,402.05,557.775, 0), v100, z5, tool0;
	MoveL Offs(p0,403.42560000000003,557.4879999999999, 0), v100, z5, tool0;
	MoveL Offs(p0,404.8348,557.2009999999999, 0), v100, z5, tool0;
	MoveL Offs(p0,406.25120000000004,556.9200000000001, 0), v100, z5, tool0;
	MoveL Offs(p0,407.64840000000004,556.6510000000001, 0), v100, z5, tool0;
	MoveL Offs(p0,409.0,556.4, 0), v100, z5, tool0;
	MoveL Offs(p0,409.0,556.4, 0), v100, z5, tool0;
	MoveJ Offs(p0,310.2,549.6, 10), v100, z1, tool0;
	MoveL Offs(p0,311.5072000000001,546.8928000000002, 0), v100, z5, tool0;
	MoveL Offs(p0,312.46979999999996,545.1881999999999, 0), v100, z5, tool0;
	MoveL Offs(p0,313.6016000000001,543.3024, 0), v100, z5, tool0;
	MoveL Offs(p0,314.875,541.275, 0), v100, z5, tool0;
	MoveL Offs(p0,316.2624,539.1456000000001, 0), v100, z5, tool0;
	MoveL Offs(p0,317.7362,536.9538, 0), v100, z5, tool0;
	MoveL Offs(p0,319.2688,534.7392, 0), v100, z5, tool0;
	MoveL Offs(p0,320.8326,532.5414000000001, 0), v100, z5, tool0;
	MoveL Offs(p0,322.4,530.4, 0), v100, z5, tool0;
	MoveL Offs(p0,323.93240000000003,528.2992000000002, 0), v100, z5, tool0;
	MoveL Offs(p0,325.39520000000005,526.2176000000001, 0), v100, z5, tool0;
	MoveL Offs(p0,326.7668,524.1863999999999, 0), v100, z5, tool0;
	MoveL Offs(p0,328.0256,522.2368, 0), v100, z5, tool0;
	MoveL Offs(p0,329.15,520.4, 0), v100, z5, tool0;
	MoveL Offs(p0,330.11839999999995,518.7072000000001, 0), v100, z5, tool0;
	MoveL Offs(p0,330.9092,517.1895999999999, 0), v100, z5, tool0;
	MoveL Offs(p0,331.5008,515.8784, 0), v100, z5, tool0;
	MoveL Offs(p0,331.8716,514.8048, 0), v100, z5, tool0;
	MoveL Offs(p0,332.0,514.0, 0), v100, z5, tool0;
	MoveL Offs(p0,331.4492,511.89219999999995, 0), v100, z5, tool0;
	MoveL Offs(p0,331.04640000000006,511.09440000000006, 0), v100, z5, tool0;
	MoveL Offs(p0,330.55,510.275, 0), v100, z5, tool0;
	MoveL Offs(p0,329.9696,509.44960000000003, 0), v100, z5, tool0;
	MoveL Offs(p0,329.3148,508.63379999999995, 0), v100, z5, tool0;
	MoveL Offs(p0,328.59520000000003,507.8432000000001, 0), v100, z5, tool0;
	MoveL Offs(p0,327.8204,507.09340000000003, 0), v100, z5, tool0;
	MoveL Offs(p0,327.0,506.4, 0), v100, z5, tool0;
	MoveL Offs(p0,324.0752000000001,503.3632000000001, 0), v100, z5, tool0;
	MoveL Offs(p0,323.1228,501.71279999999996, 0), v100, z5, tool0;
	MoveL Offs(p0,322.5136,499.9616, 0), v100, z5, tool0;
	MoveL Offs(p0,322.25,498.1, 0), v100, z5, tool0;
	MoveL Offs(p0,322.3344,496.1184, 0), v100, z5, tool0;
	MoveL Offs(p0,322.7692,494.0072, 0), v100, z5, tool0;
	MoveL Offs(p0,323.5568,491.7568000000001, 0), v100, z5, tool0;
	MoveL Offs(p0,324.69960000000003,489.3576, 0), v100, z5, tool0;
	MoveL Offs(p0,326.2,486.8, 0), v100, z5, tool0;
	MoveL Offs(p0,327.7716000000001,484.0494, 0), v100, z5, tool0;
	MoveL Offs(p0,328.8848000000001,481.54720000000015, 0), v100, z5, tool0;
	MoveL Offs(p0,329.5371999999999,479.27779999999996, 0), v100, z5, tool0;
	MoveL Offs(p0,329.7264,477.2256000000001, 0), v100, z5, tool0;
	MoveL Offs(p0,329.45,475.375, 0), v100, z5, tool0;
	MoveL Offs(p0,328.70560000000006,473.71040000000005, 0), v100, z5, tool0;
	MoveL Offs(p0,327.4908,472.2162, 0), v100, z5, tool0;
	MoveL Offs(p0,325.8032,470.8768, 0), v100, z5, tool0;
	MoveL Offs(p0,323.6404,469.67660000000006, 0), v100, z5, tool0;
	MoveL Offs(p0,321.0,468.6, 0), v100, z5, tool0;
	MoveL Offs(p0,318.87080000000003,467.90060000000005, 0), v100, z5, tool0;
	MoveL Offs(p0,317.11840000000007,467.3728000000001, 0), v100, z5, tool0;
	MoveL Offs(p0,315.6756,467.03219999999993, 0), v100, z5, tool0;
	MoveL Offs(p0,314.4752,466.8944, 0), v100, z5, tool0;
	MoveL Offs(p0,313.45,466.975, 0), v100, z5, tool0;
	MoveL Offs(p0,312.5328,467.28959999999995, 0), v100, z5, tool0;
	MoveL Offs(p0,311.6564,467.85380000000004, 0), v100, z5, tool0;
	MoveL Offs(p0,310.7536,468.68320000000006, 0), v100, z5, tool0;
	MoveL Offs(p0,309.7572,469.7934, 0), v100, z5, tool0;
	MoveL Offs(p0,308.6,471.2, 0), v100, z5, tool0;
	MoveL Offs(p0,306.72740000000005,473.879, 0), v100, z5, tool0;
	MoveL Offs(p0,305.06720000000007,476.8880000000001, 0), v100, z5, tool0;
	MoveL Offs(p0,303.6158,480.245, 0), v100, z5, tool0;
	MoveL Offs(p0,302.36960000000005,483.968, 0), v100, z5, tool0;
	MoveL Offs(p0,301.325,488.075, 0), v100, z5, tool0;
	MoveL Offs(p0,300.47839999999997,492.584, 0), v100, z5, tool0;
	MoveL Offs(p0,299.8262,497.51300000000003, 0), v100, z5, tool0;
	MoveL Offs(p0,299.3648,502.8800000000001, 0), v100, z5, tool0;
	MoveL Offs(p0,299.09060000000005,508.7030000000001, 0), v100, z5, tool0;
	MoveL Offs(p0,299.0,515.0, 0), v100, z5, tool0;
	MoveL Offs(p0,299.10960000000006,520.8622000000001, 0), v100, z5, tool0;
	MoveL Offs(p0,299.4208000000001,526.7136, 0), v100, z5, tool0;
	MoveL Offs(p0,299.9072,532.4114, 0), v100, z5, tool0;
	MoveL Offs(p0,300.5424,537.8128, 0), v100, z5, tool0;
	MoveL Offs(p0,301.3,542.775, 0), v100, z5, tool0;
	MoveL Offs(p0,302.1536,547.1551999999999, 0), v100, z5, tool0;
	MoveL Offs(p0,303.0768,550.8106, 0), v100, z5, tool0;
	MoveL Offs(p0,304.0432,553.5984000000001, 0), v100, z5, tool0;
	MoveL Offs(p0,305.0264,555.3758, 0), v100, z5, tool0;
	MoveL Offs(p0,306.0,556.0, 0), v100, z5, tool0;
	MoveL Offs(p0,308.3472,553.3216, 0), v100, z5, tool0;
	MoveL Offs(p0,308.8266,552.4818, 0), v100, z5, tool0;
	MoveL Offs(p0,309.30240000000003,551.5712000000001, 0), v100, z5, tool0;
	MoveL Offs(p0,309.7638,550.6054, 0), v100, z5, tool0;
	MoveL Offs(p0,310.2,549.6, 0), v100, z5, tool0;
	MoveL Offs(p0,310.2,549.6, 0), v100, z5, tool0;
	MoveJ Offs(p0,458.0,540.8, 10), v100, z1, tool0;
	MoveL Offs(p0,459.0064000000002,538.4112000000002, 0), v100, z5, tool0;
	MoveL Offs(p0,459.6956,537.0848, 0), v100, z5, tool0;
	MoveL Offs(p0,460.4832,535.7056000000001, 0), v100, z5, tool0;
	MoveL Offs(p0,461.35,534.3, 0), v100, z5, tool0;
	MoveL Offs(p0,462.2768,532.8944, 0), v100, z5, tool0;
	MoveL Offs(p0,463.24440000000004,531.5152, 0), v100, z5, tool0;
	MoveL Offs(p0,464.2336,530.1888000000001, 0), v100, z5, tool0;
	MoveL Offs(p0,465.22520000000003,528.9416, 0), v100, z5, tool0;
	MoveL Offs(p0,466.2,527.8, 0), v100, z5, tool0;
	MoveL Offs(p0,468.86400000000003,524.8642, 0), v100, z5, tool0;
	MoveL Offs(p0,469.62399999999997,523.9824000000001, 0), v100, z5, tool0;
	MoveL Offs(p0,470.3,523.175, 0), v100, z5, tool0;
	MoveL Offs(p0,470.88,522.4576, 0), v100, z5, tool0;
	MoveL Offs(p0,471.35200000000003,521.8458, 0), v100, z5, tool0;
	MoveL Offs(p0,471.70400000000006,521.3552000000001, 0), v100, z5, tool0;
	MoveL Offs(p0,471.924,521.0014, 0), v100, z5, tool0;
	MoveL Offs(p0,472.0,520.8, 0), v100, z5, tool0;
	MoveL Offs(p0,469.3834,518.4508, 0), v100, z5, tool0;
	MoveL Offs(p0,468.6976000000001,517.9712, 0), v100, z5, tool0;
	MoveL Offs(p0,467.9662,517.4844, 0), v100, z5, tool0;
	MoveL Offs(p0,467.2,517.0, 0), v100, z5, tool0;
	MoveL Offs(p0,464.9568000000002,515.6528000000002, 0), v100, z5, tool0;
	MoveL Offs(p0,463.97619999999995,515.2252, 0), v100, z5, tool0;
	MoveL Offs(p0,463.0304,514.9584, 0), v100, z5, tool0;
	MoveL Offs(p0,462.075,514.85, 0), v100, z5, tool0;
	MoveL Offs(p0,461.0656,514.8976, 0), v100, z5, tool0;
	MoveL Offs(p0,459.95779999999996,515.0988, 0), v100, z5, tool0;
	MoveL Offs(p0,458.7072,515.4512000000001, 0), v100, z5, tool0;
	MoveL Offs(p0,457.2694,515.9524, 0), v100, z5, tool0;
	MoveL Offs(p0,455.6,516.6, 0), v100, z5, tool0;
	MoveL Offs(p0,453.38860000000005,517.7314, 0), v100, z5, tool0;
	MoveL Offs(p0,451.0848000000002,519.1952000000001, 0), v100, z5, tool0;
	MoveL Offs(p0,448.70419999999996,520.9757999999999, 0), v100, z5, tool0;
	MoveL Offs(p0,446.26240000000007,523.0576, 0), v100, z5, tool0;
	MoveL Offs(p0,443.775,525.425, 0), v100, z5, tool0;
	MoveL Offs(p0,441.2576,528.0624, 0), v100, z5, tool0;
	MoveL Offs(p0,438.7258,530.9541999999999, 0), v100, z5, tool0;
	MoveL Offs(p0,436.1952,534.0848, 0), v100, z5, tool0;
	MoveL Offs(p0,433.68140000000005,537.4386000000001, 0), v100, z5, tool0;
	MoveL Offs(p0,431.2,541.0, 0), v100, z5, tool0;
	MoveL Offs(p0,429.0714000000001,544.3196, 0), v100, z5, tool0;
	MoveL Offs(p0,427.5152000000001,546.9888000000001, 0), v100, z5, tool0;
	MoveL Offs(p0,426.57579999999996,549.0532000000001, 0), v100, z5, tool0;
	MoveL Offs(p0,426.2976,550.5584000000001, 0), v100, z5, tool0;
	MoveL Offs(p0,426.725,551.55, 0), v100, z5, tool0;
	MoveL Offs(p0,427.90240000000006,552.0735999999999, 0), v100, z5, tool0;
	MoveL Offs(p0,429.8741999999999,552.1748, 0), v100, z5, tool0;
	MoveL Offs(p0,432.6848,551.8992000000001, 0), v100, z5, tool0;
	MoveL Offs(p0,436.3786,551.2924, 0), v100, z5, tool0;
	MoveL Offs(p0,441.0,550.4, 0), v100, z5, tool0;
	MoveL Offs(p0,444.87260000000003,549.6236000000001, 0), v100, z5, tool0;
	MoveL Offs(p0,448.02880000000016,548.9408000000001, 0), v100, z5, tool0;
	MoveL Offs(p0,450.5562,548.3011999999999, 0), v100, z5, tool0;
	MoveL Offs(p0,452.5424,547.6544000000001, 0), v100, z5, tool0;
	MoveL Offs(p0,454.075,546.95, 0), v100, z5, tool0;
	MoveL Offs(p0,455.2416,546.1376, 0), v100, z5, tool0;
	MoveL Offs(p0,456.1298,545.1668, 0), v100, z5, tool0;
	MoveL Offs(p0,456.82720000000006,543.9872, 0), v100, z5, tool0;
	MoveL Offs(p0,457.4214,542.5484, 0), v100, z5, tool0;
	MoveL Offs(p0,458.0,540.8, 0), v100, z5, tool0;
	MoveL Offs(p0,458.0,540.8, 0), v100, z5, tool0;
	MoveJ Offs(p0,730.6,488.4, 10), v100, z1, tool0;
	MoveL Offs(p0,734.7776000000001,485.8360000000001, 0), v100, z5, tool0;
	MoveL Offs(p0,738.6768000000002,482.93600000000004, 0), v100, z5, tool0;
	MoveL Offs(p0,742.3072,479.68799999999993, 0), v100, z5, tool0;
	MoveL Offs(p0,745.6784,476.0800000000001, 0), v100, z5, tool0;
	MoveL Offs(p0,748.8,472.1, 0), v100, z5, tool0;
	MoveL Offs(p0,751.6816,467.736, 0), v100, z5, tool0;
	MoveL Offs(p0,754.3328,462.97599999999994, 0), v100, z5, tool0;
	MoveL Offs(p0,756.7632000000001,457.808, 0), v100, z5, tool0;
	MoveL Offs(p0,758.9824000000001,452.21999999999997, 0), v100, z5, tool0;
	MoveL Offs(p0,761.0,446.2, 0), v100, z5, tool0;
	MoveL Offs(p0,765.9480000000001,430.7050000000001, 0), v100, z5, tool0;
	MoveL Offs(p0,770.7760000000003,416.9920000000001, 0), v100, z5, tool0;
	MoveL Offs(p0,775.5799999999999,404.899, 0), v100, z5, tool0;
	MoveL Offs(p0,780.4559999999999,394.26400000000007, 0), v100, z5, tool0;
	MoveL Offs(p0,785.5,384.925, 0), v100, z5, tool0;
	MoveL Offs(p0,790.8079999999999,376.71999999999997, 0), v100, z5, tool0;
	MoveL Offs(p0,796.476,369.48699999999997, 0), v100, z5, tool0;
	MoveL Offs(p0,802.6000000000001,363.064, 0), v100, z5, tool0;
	MoveL Offs(p0,809.2760000000001,357.28900000000004, 0), v100, z5, tool0;
	MoveL Offs(p0,816.6,352.0, 0), v100, z5, tool0;
	MoveL Offs(p0,822.5716000000002,348.36480000000006, 0), v100, z5, tool0;
	MoveL Offs(p0,828.8288,345.26240000000007, 0), v100, z5, tool0;
	MoveL Offs(p0,835.3452,342.69759999999997, 0), v100, z5, tool0;
	MoveL Offs(p0,842.0944000000002,340.6752, 0), v100, z5, tool0;
	MoveL Offs(p0,849.05,339.2, 0), v100, z5, tool0;
	MoveL Offs(p0,856.1856,338.2768, 0), v100, z5, tool0;
	MoveL Offs(p0,863.4748,337.91040000000004, 0), v100, z5, tool0;
	MoveL Offs(p0,870.8912,338.10560000000004, 0), v100, z5, tool0;
	MoveL Offs(p0,878.4084,338.8672, 0), v100, z5, tool0;
	MoveL Offs(p0,886.0,340.2, 0), v100, z5, tool0;
	MoveL Offs(p0,894.5142,342.71220000000005, 0), v100, z5, tool0;
	MoveL Offs(p0,902.1296000000002,346.3296000000001, 0), v100, z5, tool0;
	MoveL Offs(p0,908.7754000000001,350.9334, 0), v100, z5, tool0;
	MoveL Offs(p0,914.3808000000001,356.4048, 0), v100, z5, tool0;
	MoveL Offs(p0,918.875,362.625, 0), v100, z5, tool0;
	MoveL Offs(p0,922.1872,369.4752, 0), v100, z5, tool0;
	MoveL Offs(p0,924.2466000000001,376.8366, 0), v100, z5, tool0;
	MoveL Offs(p0,924.9824000000001,384.59040000000005, 0), v100, z5, tool0;
	MoveL Offs(p0,924.3238000000001,392.6178, 0), v100, z5, tool0;
	MoveL Offs(p0,922.2,400.8, 0), v100, z5, tool0;
	MoveL Offs(p0,917.9613999999999,410.5964, 0), v100, z5, tool0;
	MoveL Offs(p0,912.4112000000002,419.65120000000013, 0), v100, z5, tool0;
	MoveL Offs(p0,905.6777999999998,427.8828, 0), v100, z5, tool0;
	MoveL Offs(p0,897.8896000000001,435.20959999999997, 0), v100, z5, tool0;
	MoveL Offs(p0,889.175,441.55, 0), v100, z5, tool0;
	MoveL Offs(p0,879.6623999999999,446.8224, 0), v100, z5, tool0;
	MoveL Offs(p0,869.4802,450.9452, 0), v100, z5, tool0;
	MoveL Offs(p0,858.7567999999999,453.83680000000004, 0), v100, z5, tool0;
	MoveL Offs(p0,847.6206,455.4156, 0), v100, z5, tool0;
	MoveL Offs(p0,836.2,455.6, 0), v100, z5, tool0;
	MoveL Offs(p0,833.1458,455.5042, 0), v100, z5, tool0;
	MoveL Offs(p0,830.4624000000001,455.4576000000002, 0), v100, z5, tool0;
	MoveL Offs(p0,828.1485999999999,455.46139999999997, 0), v100, z5, tool0;
	MoveL Offs(p0,826.2032000000002,455.51680000000005, 0), v100, z5, tool0;
	MoveL Offs(p0,824.625,455.625, 0), v100, z5, tool0;
	MoveL Offs(p0,823.4128000000001,455.78720000000004, 0), v100, z5, tool0;
	MoveL Offs(p0,822.5654000000001,456.00460000000004, 0), v100, z5, tool0;
	MoveL Offs(p0,822.0816000000001,456.27840000000003, 0), v100, z5, tool0;
	MoveL Offs(p0,821.9602000000001,456.6098, 0), v100, z5, tool0;
	MoveL Offs(p0,822.2,457.0, 0), v100, z5, tool0;
	MoveL Offs(p0,825.4652,457.87299999999993, 0), v100, z5, tool0;
	MoveL Offs(p0,827.4703999999999,458.1360000000001, 0), v100, z5, tool0;
	MoveL Offs(p0,829.85,458.375, 0), v100, z5, tool0;
	MoveL Offs(p0,832.5536,458.584, 0), v100, z5, tool0;
	MoveL Offs(p0,835.5308000000001,458.75699999999995, 0), v100, z5, tool0;
	MoveL Offs(p0,838.7312,458.88800000000003, 0), v100, z5, tool0;
	MoveL Offs(p0,842.1044000000002,458.9710000000001, 0), v100, z5, tool0;
	MoveL Offs(p0,845.6,459.0, 0), v100, z5, tool0;
	MoveL Offs(p0,851.3304,458.9862000000001, 0), v100, z5, tool0;
	MoveL Offs(p0,856.0672000000002,458.91360000000014, 0), v100, z5, tool0;
	MoveL Offs(p0,860.0288,458.7354, 0), v100, z5, tool0;
	MoveL Offs(p0,863.4336000000001,458.4048000000001, 0), v100, z5, tool0;
	MoveL Offs(p0,866.5,457.875, 0), v100, z5, tool0;
	MoveL Offs(p0,869.4464,457.0992, 0), v100, z5, tool0;
	MoveL Offs(p0,872.4912,456.03060000000005, 0), v100, z5, tool0;
	MoveL Offs(p0,875.8528000000002,454.6224, 0), v100, z5, tool0;
	MoveL Offs(p0,879.7495999999999,452.8278, 0), v100, z5, tool0;
	MoveL Offs(p0,884.4,450.6, 0), v100, z5, tool0;
	MoveL Offs(p0,890.3076000000001,447.58459999999997, 0), v100, z5, tool0;
	MoveL Offs(p0,895.8048000000005,444.4048000000001, 0), v100, z5, tool0;
	MoveL Offs(p0,900.9132,441.0402, 0), v100, z5, tool0;
	MoveL Offs(p0,905.6544000000001,437.4704, 0), v100, z5, tool0;
	MoveL Offs(p0,910.05,433.675, 0), v100, z5, tool0;
	MoveL Offs(p0,914.1216000000001,429.6336, 0), v100, z5, tool0;
	MoveL Offs(p0,917.8907999999999,425.32579999999996, 0), v100, z5, tool0;
	MoveL Offs(p0,921.3792000000001,420.7312, 0), v100, z5, tool0;
	MoveL Offs(p0,924.6084000000001,415.82939999999996, 0), v100, z5, tool0;
	MoveL Offs(p0,927.6,410.6, 0), v100, z5, tool0;
	MoveL Offs(p0,929.8682000000001,405.99940000000004, 0), v100, z5, tool0;
	MoveL Offs(p0,931.7536000000002,401.5392000000001, 0), v100, z5, tool0;
	MoveL Offs(p0,933.2573999999998,397.1918, 0), v100, z5, tool0;
	MoveL Offs(p0,934.3808000000001,392.92960000000005, 0), v100, z5, tool0;
	MoveL Offs(p0,935.125,388.725, 0), v100, z5, tool0;
	MoveL Offs(p0,935.4912,384.55039999999997, 0), v100, z5, tool0;
	MoveL Offs(p0,935.4805999999999,380.3782, 0), v100, z5, tool0;
	MoveL Offs(p0,935.0944,376.18080000000003, 0), v100, z5, tool0;
	MoveL Offs(p0,934.3338,371.9306, 0), v100, z5, tool0;
	MoveL Offs(p0,933.2,367.6, 0), v100, z5, tool0;
	MoveL Offs(p0,931.7818000000001,363.3858000000001, 0), v100, z5, tool0;
	MoveL Offs(p0,929.9424000000002,359.2784000000001, 0), v100, z5, tool0;
	MoveL Offs(p0,927.7045999999998,355.3005999999999, 0), v100, z5, tool0;
	MoveL Offs(p0,925.0912000000001,351.4752, 0), v100, z5, tool0;
	MoveL Offs(p0,922.125,347.825, 0), v100, z5, tool0;
	MoveL Offs(p0,918.8287999999999,344.3728, 0), v100, z5, tool0;
	MoveL Offs(p0,915.2254,341.1414, 0), v100, z5, tool0;
	MoveL Offs(p0,911.3376000000001,338.1536, 0), v100, z5, tool0;
	MoveL Offs(p0,907.1882000000002,335.4322, 0), v100, z5, tool0;
	MoveL Offs(p0,902.8,333.0, 0), v100, z5, tool0;
	MoveL Offs(p0,899.9014000000001,331.56780000000003, 0), v100, z5, tool0;
	MoveL Offs(p0,897.2512,330.3744000000001, 0), v100, z5, tool0;
	MoveL Offs(p0,894.7378000000001,329.39459999999997, 0), v100, z5, tool0;
	MoveL Offs(p0,892.2496000000001,328.6032000000001, 0), v100, z5, tool0;
	MoveL Offs(p0,889.675,327.975, 0), v100, z5, tool0;
	MoveL Offs(p0,886.9024,327.4848, 0), v100, z5, tool0;
	MoveL Offs(p0,883.8202000000001,327.1074, 0), v100, z5, tool0;
	MoveL Offs(p0,880.3168000000002,326.8176, 0), v100, z5, tool0;
	MoveL Offs(p0,876.2806,326.5902, 0), v100, z5, tool0;
	MoveL Offs(p0,871.6,326.4, 0), v100, z5, tool0;
	MoveL Offs(p0,867.1398000000002,326.2576, 0), v100, z5, tool0;
	MoveL Offs(p0,863.1824000000003,326.19680000000005, 0), v100, z5, tool0;
	MoveL Offs(p0,859.6426000000001,326.2272, 0), v100, z5, tool0;
	MoveL Offs(p0,856.4352000000001,326.3584, 0), v100, z5, tool0;
	MoveL Offs(p0,853.475,326.6, 0), v100, z5, tool0;
	MoveL Offs(p0,850.6768,326.9616, 0), v100, z5, tool0;
	MoveL Offs(p0,847.9554,327.4527999999999, 0), v100, z5, tool0;
	MoveL Offs(p0,845.2256000000001,328.08320000000003, 0), v100, z5, tool0;
	MoveL Offs(p0,842.4022000000001,328.8624, 0), v100, z5, tool0;
	MoveL Offs(p0,839.4,329.8, 0), v100, z5, tool0;
	MoveL Offs(p0,827.3848000000002,334.49660000000006, 0), v100, z5, tool0;
	MoveL Offs(p0,816.2624000000003,340.2288000000001, 0), v100, z5, tool0;
	MoveL Offs(p0,805.9775999999999,347.06019999999995, 0), v100, z5, tool0;
	MoveL Offs(p0,796.4752000000001,355.0544, 0), v100, z5, tool0;
	MoveL Offs(p0,787.7,364.275, 0), v100, z5, tool0;
	MoveL Offs(p0,779.5968,374.78560000000004, 0), v100, z5, tool0;
	MoveL Offs(p0,772.1103999999999,386.6498, 0), v100, z5, tool0;
	MoveL Offs(p0,765.1856,399.9312000000001, 0), v100, z5, tool0;
	MoveL Offs(p0,758.7672,414.6934, 0), v100, z5, tool0;
	MoveL Offs(p0,752.8,431.0, 0), v100, z5, tool0;
	MoveL Offs(p0,751.5796,434.6740000000001, 0), v100, z5, tool0;
	MoveL Offs(p0,750.3328,438.3360000000001, 0), v100, z5, tool0;
	MoveL Offs(p0,749.0812,441.92599999999993, 0), v100, z5, tool0;
	MoveL Offs(p0,747.8464,445.384, 0), v100, z5, tool0;
	MoveL Offs(p0,746.65,448.65, 0), v100, z5, tool0;
	MoveL Offs(p0,745.5136,451.66399999999993, 0), v100, z5, tool0;
	MoveL Offs(p0,744.4588,454.366, 0), v100, z5, tool0;
	MoveL Offs(p0,743.5072,456.6960000000001, 0), v100, z5, tool0;
	MoveL Offs(p0,742.6804,458.59400000000005, 0), v100, z5, tool0;
	MoveL Offs(p0,742.0,460.0, 0), v100, z5, tool0;
	MoveL Offs(p0,738.3943999999999,465.8604, 0), v100, z5, tool0;
	MoveL Offs(p0,734.0112000000001,471.05120000000016, 0), v100, z5, tool0;
	MoveL Offs(p0,728.9608000000001,475.5268, 0), v100, z5, tool0;
	MoveL Offs(p0,723.3536000000001,479.2416, 0), v100, z5, tool0;
	MoveL Offs(p0,717.3,482.15, 0), v100, z5, tool0;
	MoveL Offs(p0,710.9104,484.20640000000003, 0), v100, z5, tool0;
	MoveL Offs(p0,704.2951999999999,485.3652, 0), v100, z5, tool0;
	MoveL Offs(p0,697.5648000000001,485.58080000000007, 0), v100, z5, tool0;
	MoveL Offs(p0,690.8296,484.8076, 0), v100, z5, tool0;
	MoveL Offs(p0,684.2,483.0, 0), v100, z5, tool0;
	MoveL Offs(p0,676.0,480.2, 0), v100, z5, tool0;
	MoveL Offs(p0,676.0,486.0, 0), v100, z5, tool0;
	MoveL Offs(p0,676.1680000000001,488.40480000000014, 0), v100, z5, tool0;
	MoveL Offs(p0,676.405,489.3731999999999, 0), v100, z5, tool0;
	MoveL Offs(p0,676.768,490.2144, 0), v100, z5, tool0;
	MoveL Offs(p0,677.275,490.95, 0), v100, z5, tool0;
	MoveL Offs(p0,677.9440000000001,491.60159999999996, 0), v100, z5, tool0;
	MoveL Offs(p0,678.793,492.19079999999997, 0), v100, z5, tool0;
	MoveL Offs(p0,679.8399999999999,492.7392000000001, 0), v100, z5, tool0;
	MoveL Offs(p0,681.1030000000001,493.26840000000004, 0), v100, z5, tool0;
	MoveL Offs(p0,682.6,493.8, 0), v100, z5, tool0;
	MoveL Offs(p0,687.3352,495.0906000000001, 0), v100, z5, tool0;
	MoveL Offs(p0,692.1616000000002,495.9648000000001, 0), v100, z5, tool0;
	MoveL Offs(p0,697.0503999999999,496.42620000000005, 0), v100, z5, tool0;
	MoveL Offs(p0,701.9728,496.4784000000001, 0), v100, z5, tool0;
	MoveL Offs(p0,706.9,496.125, 0), v100, z5, tool0;
	MoveL Offs(p0,711.8032,495.3696, 0), v100, z5, tool0;
	MoveL Offs(p0,716.6536,494.21579999999994, 0), v100, z5, tool0;
	MoveL Offs(p0,721.4224,492.66720000000004, 0), v100, z5, tool0;
	MoveL Offs(p0,726.0808,490.72740000000005, 0), v100, z5, tool0;
	MoveL Offs(p0,730.6,488.4, 0), v100, z5, tool0;
	MoveL Offs(p0,730.6,488.4, 0), v100, z5, tool0;
	MoveJ Offs(p0,402.6,477.8, 10), v100, z1, tool0;
	MoveL Offs(p0,406.2720000000001,475.48480000000006, 0), v100, z5, tool0;
	MoveL Offs(p0,408.32399999999996,473.9462, 0), v100, z5, tool0;
	MoveL Offs(p0,410.424,472.23840000000007, 0), v100, z5, tool0;
	MoveL Offs(p0,412.5,470.425, 0), v100, z5, tool0;
	MoveL Offs(p0,414.48,468.5696, 0), v100, z5, tool0;
	MoveL Offs(p0,416.29200000000003,466.73580000000004, 0), v100, z5, tool0;
	MoveL Offs(p0,417.86400000000003,464.98720000000003, 0), v100, z5, tool0;
	MoveL Offs(p0,419.12399999999997,463.38739999999996, 0), v100, z5, tool0;
	MoveL Offs(p0,420.0,462.0, 0), v100, z5, tool0;
	MoveL Offs(p0,419.40160000000003,459.85920000000004, 0), v100, z5, tool0;
	MoveL Offs(p0,418.325,459.6, 0), v100, z5, tool0;
	MoveL Offs(p0,416.77439999999996,459.43680000000006, 0), v100, z5, tool0;
	MoveL Offs(p0,414.6982,459.3624, 0), v100, z5, tool0;
	MoveL Offs(p0,412.0448,459.3696, 0), v100, z5, tool0;
	MoveL Offs(p0,408.7626,459.4512000000001, 0), v100, z5, tool0;
	MoveL Offs(p0,404.8,459.6, 0), v100, z5, tool0;
	MoveL Offs(p0,396.7316,459.6924000000001, 0), v100, z5, tool0;
	MoveL Offs(p0,388.3008000000001,459.35520000000014, 0), v100, z5, tool0;
	MoveL Offs(p0,379.40919999999994,458.56680000000006, 0), v100, z5, tool0;
	MoveL Offs(p0,369.95840000000004,457.3056, 0), v100, z5, tool0;
	MoveL Offs(p0,359.85,455.55, 0), v100, z5, tool0;
	MoveL Offs(p0,348.9856,453.2784, 0), v100, z5, tool0;
	MoveL Offs(p0,337.2668,450.4692, 0), v100, z5, tool0;
	MoveL Offs(p0,324.59520000000003,447.1008, 0), v100, z5, tool0;
	MoveL Offs(p0,310.8724,443.1516, 0), v100, z5, tool0;
	MoveL Offs(p0,296.0,438.6, 0), v100, z5, tool0;
	MoveL Offs(p0,282.70720000000006,434.2808000000001, 0), v100, z5, tool0;
	MoveL Offs(p0,269.16960000000006,429.5584000000002, 0), v100, z5, tool0;
	MoveL Offs(p0,255.65839999999997,424.5455999999999, 0), v100, z5, tool0;
	MoveL Offs(p0,242.44480000000004,419.3552000000001, 0), v100, z5, tool0;
	MoveL Offs(p0,229.8,414.1, 0), v100, z5, tool0;
	MoveL Offs(p0,217.99519999999998,408.89279999999997, 0), v100, z5, tool0;
	MoveL Offs(p0,207.30159999999995,403.8464, 0), v100, z5, tool0;
	MoveL Offs(p0,197.99040000000002,399.0736, 0), v100, z5, tool0;
	MoveL Offs(p0,190.3328,394.6872, 0), v100, z5, tool0;
	MoveL Offs(p0,184.6,390.8, 0), v100, z5, tool0;
	MoveL Offs(p0,180.96320000000006,388.26240000000007, 0), v100, z5, tool0;
	MoveL Offs(p0,179.3998,387.3476, 0), v100, z5, tool0;
	MoveL Offs(p0,178.01760000000002,386.6752, 0), v100, z5, tool0;
	MoveL Offs(p0,176.825,386.25, 0), v100, z5, tool0;
	MoveL Offs(p0,175.8304,386.0768, 0), v100, z5, tool0;
	MoveL Offs(p0,175.0422,386.16040000000004, 0), v100, z5, tool0;
	MoveL Offs(p0,174.46880000000002,386.5056000000001, 0), v100, z5, tool0;
	MoveL Offs(p0,174.11860000000001,387.1172, 0), v100, z5, tool0;
	MoveL Offs(p0,174.0,388.0, 0), v100, z5, tool0;
	MoveL Offs(p0,171.6672,389.9764, 0), v100, z5, tool0;
	MoveL Offs(p0,171.2,390.0, 0), v100, z5, tool0;
	MoveL Offs(p0,169.08480000000006,390.65120000000013, 0), v100, z5, tool0;
	MoveL Offs(p0,168.2642,391.38779999999997, 0), v100, z5, tool0;
	MoveL Offs(p0,167.62240000000003,392.3296, 0), v100, z5, tool0;
	MoveL Offs(p0,167.175,393.425, 0), v100, z5, tool0;
	MoveL Offs(p0,166.9376,394.6224, 0), v100, z5, tool0;
	MoveL Offs(p0,166.92579999999998,395.87019999999995, 0), v100, z5, tool0;
	MoveL Offs(p0,167.1552,397.11680000000007, 0), v100, z5, tool0;
	MoveL Offs(p0,167.64140000000003,398.31059999999997, 0), v100, z5, tool0;
	MoveL Offs(p0,168.4,399.4, 0), v100, z5, tool0;
	MoveL Offs(p0,173.35240000000005,403.216, 0), v100, z5, tool0;
	MoveL Offs(p0,182.81920000000005,408.4720000000001, 0), v100, z5, tool0;
	MoveL Offs(p0,196.0948,414.88, 0), v100, z5, tool0;
	MoveL Offs(p0,212.47359999999998,422.15200000000004, 0), v100, z5, tool0;
	MoveL Offs(p0,231.25,430.0, 0), v100, z5, tool0;
	MoveL Offs(p0,251.71840000000003,438.13599999999997, 0), v100, z5, tool0;
	MoveL Offs(p0,273.1732,446.27200000000005, 0), v100, z5, tool0;
	MoveL Offs(p0,294.90880000000004,454.12000000000006, 0), v100, z5, tool0;
	MoveL Offs(p0,316.2196,461.392, 0), v100, z5, tool0;
	MoveL Offs(p0,336.4,467.8, 0), v100, z5, tool0;
	MoveL Offs(p0,347.7198,471.17420000000004, 0), v100, z5, tool0;
	MoveL Offs(p0,357.7424000000001,473.98560000000015, 0), v100, z5, tool0;
	MoveL Offs(p0,366.56260000000003,476.2474, 0), v100, z5, tool0;
	MoveL Offs(p0,374.27520000000004,477.9728000000001, 0), v100, z5, tool0;
	MoveL Offs(p0,380.975,479.175, 0), v100, z5, tool0;
	MoveL Offs(p0,386.7568,479.86719999999997, 0), v100, z5, tool0;
	MoveL Offs(p0,391.71540000000005,480.06260000000003, 0), v100, z5, tool0;
	MoveL Offs(p0,395.9456,479.77440000000007, 0), v100, z5, tool0;
	MoveL Offs(p0,399.5422,479.0158, 0), v100, z5, tool0;
	MoveL Offs(p0,402.6,477.8, 0), v100, z5, tool0;
	MoveL Offs(p0,402.6,477.8, 0), v100, z5, tool0;
	MoveJ Offs(p0,336.8,476.2, 10), v100, z1, tool0;
	MoveL Offs(p0,336.20779999999996,474.01180000000005, 0), v100, z5, tool0;
	MoveL Offs(p0,335.85920000000004,473.7232, 0), v100, z5, tool0;
	MoveL Offs(p0,335.4554,473.4514000000001, 0), v100, z5, tool0;
	MoveL Offs(p0,335.0,473.2, 0), v100, z5, tool0;
	MoveL Offs(p0,332.825,473.2, 0), v100, z5, tool0;
	MoveL Offs(p0,332.5376,473.416, 0), v100, z5, tool0;
	MoveL Offs(p0,332.3078,473.704, 0), v100, z5, tool0;
	MoveL Offs(p0,332.1392,474.064, 0), v100, z5, tool0;
	MoveL Offs(p0,332.03540000000004,474.496, 0), v100, z5, tool0;
	MoveL Offs(p0,332.0,475.0, 0), v100, z5, tool0;
	MoveL Offs(p0,332.73440000000005,477.1995999999999, 0), v100, z5, tool0;
	MoveL Offs(p0,333.22880000000004,477.6112, 0), v100, z5, tool0;
	MoveL Offs(p0,333.8,477.85, 0), v100, z5, tool0;
	MoveL Offs(p0,334.4192,477.9088, 0), v100, z5, tool0;
	MoveL Offs(p0,335.0576,477.7804, 0), v100, z5, tool0;
	MoveL Offs(p0,335.68640000000005,477.45760000000007, 0), v100, z5, tool0;
	MoveL Offs(p0,336.2768,476.93320000000006, 0), v100, z5, tool0;
	MoveL Offs(p0,336.8,476.2, 0), v100, z5, tool0;
	MoveL Offs(p0,336.8,476.2, 0), v100, z5, tool0;
	MoveJ Offs(p0,103.4,450.6, 10), v100, z1, tool0;
	MoveL Offs(p0,105.91040000000002,449.1632000000001, 0), v100, z5, tool0;
	MoveL Offs(p0,107.2106,448.29779999999994, 0), v100, z5, tool0;
	MoveL Offs(p0,108.50720000000001,447.3616, 0), v100, z5, tool0;
	MoveL Offs(p0,109.775,446.375, 0), v100, z5, tool0;
	MoveL Offs(p0,110.9888,445.35839999999996, 0), v100, z5, tool0;
	MoveL Offs(p0,112.12339999999999,444.3322, 0), v100, z5, tool0;
	MoveL Offs(p0,113.15360000000001,443.31680000000006, 0), v100, z5, tool0;
	MoveL Offs(p0,114.0542,442.3326, 0), v100, z5, tool0;
	MoveL Offs(p0,114.8,441.4, 0), v100, z5, tool0;
	MoveL Offs(p0,117.0258,437.26620000000014, 0), v100, z5, tool0;
	MoveL Offs(p0,118.44640000000004,432.08960000000013, 0), v100, z5, tool0;
	MoveL Offs(p0,119.0966,426.0874, 0), v100, z5, tool0;
	MoveL Offs(p0,119.0112,419.4768, 0), v100, z5, tool0;
	MoveL Offs(p0,118.225,412.475, 0), v100, z5, tool0;
	MoveL Offs(p0,116.7728,405.2992, 0), v100, z5, tool0;
	MoveL Offs(p0,114.6894,398.16659999999996, 0), v100, z5, tool0;
	MoveL Offs(p0,112.0096,391.29440000000005, 0), v100, z5, tool0;
	MoveL Offs(p0,108.76820000000001,384.8998, 0), v100, z5, tool0;
	MoveL Offs(p0,105.0,379.2, 0), v100, z5, tool0;
	MoveL Offs(p0,102.16499999999999,377.04900000000004, 0), v100, z5, tool0;
	MoveL Offs(p0,101.24000000000001,376.88, 0), v100, z5, tool0;
	MoveL Offs(p0,100.375,376.975, 0), v100, z5, tool0;
	MoveL Offs(p0,99.6,377.32800000000003, 0), v100, z5, tool0;
	MoveL Offs(p0,98.94500000000001,377.933, 0), v100, z5, tool0;
	MoveL Offs(p0,98.44000000000001,378.784, 0), v100, z5, tool0;
	MoveL Offs(p0,98.11500000000001,379.875, 0), v100, z5, tool0;
	MoveL Offs(p0,98.0,381.2, 0), v100, z5, tool0;
	MoveL Offs(p0,97.2062,383.31319999999994, 0), v100, z5, tool0;
	MoveL Offs(p0,96.63040000000001,384.32640000000004, 0), v100, z5, tool0;
	MoveL Offs(p0,95.925,385.45, 0), v100, z5, tool0;
	MoveL Offs(p0,95.1056,386.6576, 0), v100, z5, tool0;
	MoveL Offs(p0,94.1878,387.9228, 0), v100, z5, tool0;
	MoveL Offs(p0,93.1872,389.21920000000006, 0), v100, z5, tool0;
	MoveL Offs(p0,92.11940000000001,390.5204, 0), v100, z5, tool0;
	MoveL Offs(p0,91.0,391.8, 0), v100, z5, tool0;
	MoveL Offs(p0,88.49320000000002,394.26340000000005, 0), v100, z5, tool0;
	MoveL Offs(p0,85.68160000000003,396.4832000000001, 0), v100, z5, tool0;
	MoveL Offs(p0,82.60839999999999,398.4438, 0), v100, z5, tool0;
	MoveL Offs(p0,79.3168,400.12960000000004, 0), v100, z5, tool0;
	MoveL Offs(p0,75.85,401.525, 0), v100, z5, tool0;
	MoveL Offs(p0,72.25119999999998,402.6144, 0), v100, z5, tool0;
	MoveL Offs(p0,68.5636,403.3822, 0), v100, z5, tool0;
	MoveL Offs(p0,64.83040000000001,403.81280000000004, 0), v100, z5, tool0;
	MoveL Offs(p0,61.0948,403.89060000000006, 0), v100, z5, tool0;
	MoveL Offs(p0,57.4,403.6, 0), v100, z5, tool0;
	MoveL Offs(p0,50.8,402.8, 0), v100, z5, tool0;
	MoveL Offs(p0,55.6,416.0, 0), v100, z5, tool0;
	MoveL Offs(p0,56.45180000000001,418.4456, 0), v100, z5, tool0;
	MoveL Offs(p0,57.206400000000016,420.8528000000001, 0), v100, z5, tool0;
	MoveL Offs(p0,57.862599999999986,423.2072, 0), v100, z5, tool0;
	MoveL Offs(p0,58.419200000000004,425.49440000000004, 0), v100, z5, tool0;
	MoveL Offs(p0,58.875,427.7, 0), v100, z5, tool0;
	MoveL Offs(p0,59.2288,429.80959999999993, 0), v100, z5, tool0;
	MoveL Offs(p0,59.47940000000001,431.80879999999996, 0), v100, z5, tool0;
	MoveL Offs(p0,59.625600000000006,433.68320000000006, 0), v100, z5, tool0;
	MoveL Offs(p0,59.6662,435.4184, 0), v100, z5, tool0;
	MoveL Offs(p0,59.6,437.0, 0), v100, z5, tool0;
	MoveL Offs(p0,59.40320000000003,440.45600000000013, 0), v100, z5, tool0;
	MoveL Offs(p0,59.44879999999999,441.86, 0), v100, z5, tool0;
	MoveL Offs(p0,59.6096,443.096, 0), v100, z5, tool0;
	MoveL Offs(p0,59.9,444.2, 0), v100, z5, tool0;
	MoveL Offs(p0,60.3344,445.20799999999997, 0), v100, z5, tool0;
	MoveL Offs(p0,60.92719999999999,446.15600000000006, 0), v100, z5, tool0;
	MoveL Offs(p0,61.69280000000001,447.0800000000001, 0), v100, z5, tool0;
	MoveL Offs(p0,62.6456,448.01599999999996, 0), v100, z5, tool0;
	MoveL Offs(p0,63.8,449.0, 0), v100, z5, tool0;
	MoveL Offs(p0,66.37219999999999,450.9853999999999, 0), v100, z5, tool0;
	MoveL Offs(p0,67.2784,451.62080000000003, 0), v100, z5, tool0;
	MoveL Offs(p0,68.175,452.225, 0), v100, z5, tool0;
	MoveL Offs(p0,69.0416,452.78720000000004, 0), v100, z5, tool0;
	MoveL Offs(p0,69.8578,453.29659999999996, 0), v100, z5, tool0;
	MoveL Offs(p0,70.6032,453.7424000000001, 0), v100, z5, tool0;
	MoveL Offs(p0,71.2574,454.11379999999997, 0), v100, z5, tool0;
	MoveL Offs(p0,71.8,454.4, 0), v100, z5, tool0;
	MoveL Offs(p0,76.23840000000004,455.31040000000013, 0), v100, z5, tool0;
	MoveL Offs(p0,79.3186,455.39360000000005, 0), v100, z5, tool0;
	MoveL Offs(p0,82.7792,455.25120000000004, 0), v100, z5, tool0;
	MoveL Offs(p0,86.475,454.9, 0), v100, z5, tool0;
	MoveL Offs(p0,90.26079999999999,454.3568, 0), v100, z5, tool0;
	MoveL Offs(p0,93.9914,453.6384, 0), v100, z5, tool0;
	MoveL Offs(p0,97.5216,452.7616, 0), v100, z5, tool0;
	MoveL Offs(p0,100.7062,451.7432, 0), v100, z5, tool0;
	MoveL Offs(p0,103.4,450.6, 0), v100, z5, tool0;
	MoveL Offs(p0,103.4,450.6, 0), v100, z5, tool0;
	MoveJ Offs(p0,421.6,454.8, 10), v100, z1, tool0;
	MoveL Offs(p0,424.6224000000001,453.28160000000014, 0), v100, z5, tool0;
	MoveL Offs(p0,425.4286,452.2134, 0), v100, z5, tool0;
	MoveL Offs(p0,425.76320000000004,450.95680000000004, 0), v100, z5, tool0;
	MoveL Offs(p0,425.625,449.525, 0), v100, z5, tool0;
	MoveL Offs(p0,425.01279999999997,447.9312, 0), v100, z5, tool0;
	MoveL Offs(p0,423.92539999999997,446.18860000000006, 0), v100, z5, tool0;
	MoveL Offs(p0,422.3616,444.3104, 0), v100, z5, tool0;
	MoveL Offs(p0,420.3202,442.3098, 0), v100, z5, tool0;
	MoveL Offs(p0,417.8,440.2, 0), v100, z5, tool0;
	MoveL Offs(p0,415.6838000000001,438.44980000000004, 0), v100, z5, tool0;
	MoveL Offs(p0,413.9984000000001,436.9984000000001, 0), v100, z5, tool0;
	MoveL Offs(p0,412.7186,435.78459999999995, 0), v100, z5, tool0;
	MoveL Offs(p0,411.8192,434.74719999999996, 0), v100, z5, tool0;
	MoveL Offs(p0,411.275,433.825, 0), v100, z5, tool0;
	MoveL Offs(p0,411.06080000000003,432.95680000000004, 0), v100, z5, tool0;
	MoveL Offs(p0,411.1514,432.08140000000003, 0), v100, z5, tool0;
	MoveL Offs(p0,411.52160000000003,431.1376, 0), v100, z5, tool0;
	MoveL Offs(p0,412.1462,430.06419999999997, 0), v100, z5, tool0;
	MoveL Offs(p0,413.0,428.8, 0), v100, z5, tool0;
	MoveL Offs(p0,414.5660000000001,426.02799999999996, 0), v100, z5, tool0;
	MoveL Offs(p0,414.82399999999996,425.36, 0), v100, z5, tool0;
	MoveL Offs(p0,414.95,424.8, 0), v100, z5, tool0;
	MoveL Offs(p0,414.94399999999996,424.33599999999996, 0), v100, z5, tool0;
	MoveL Offs(p0,414.8059999999999,423.95599999999996, 0), v100, z5, tool0;
	MoveL Offs(p0,414.53600000000006,423.648, 0), v100, z5, tool0;
	MoveL Offs(p0,414.134,423.4, 0), v100, z5, tool0;
	MoveL Offs(p0,413.6,423.2, 0), v100, z5, tool0;
	MoveL Offs(p0,399.62739999999997,418.76100000000014, 0), v100, z5, tool0;
	MoveL Offs(p0,386.2032000000001,413.8720000000001, 0), v100, z5, tool0;
	MoveL Offs(p0,373.40779999999995,408.57499999999993, 0), v100, z5, tool0;
	MoveL Offs(p0,361.32160000000005,402.91200000000003, 0), v100, z5, tool0;
	MoveL Offs(p0,350.025,396.925, 0), v100, z5, tool0;
	MoveL Offs(p0,339.5984,390.65599999999995, 0), v100, z5, tool0;
	MoveL Offs(p0,330.12219999999996,384.14700000000005, 0), v100, z5, tool0;
	MoveL Offs(p0,321.6768,377.44000000000005, 0), v100, z5, tool0;
	MoveL Offs(p0,314.34260000000006,370.577, 0), v100, z5, tool0;
	MoveL Offs(p0,308.2,363.6, 0), v100, z5, tool0;
	MoveL Offs(p0,304.612,358.9732, 0), v100, z5, tool0;
	MoveL Offs(p0,302.10400000000004,355.40960000000007, 0), v100, z5, tool0;
	MoveL Offs(p0,300.64,352.9044, 0), v100, z5, tool0;
	MoveL Offs(p0,300.1840000000001,351.4528, 0), v100, z5, tool0;
	MoveL Offs(p0,300.7,351.05, 0), v100, z5, tool0;
	MoveL Offs(p0,302.152,351.6912, 0), v100, z5, tool0;
	MoveL Offs(p0,304.504,353.37159999999994, 0), v100, z5, tool0;
	MoveL Offs(p0,307.7200000000001,356.0864, 0), v100, z5, tool0;
	MoveL Offs(p0,311.764,359.8308, 0), v100, z5, tool0;
	MoveL Offs(p0,316.6,364.6, 0), v100, z5, tool0;
	MoveL Offs(p0,322.216,370.0738, 0), v100, z5, tool0;
	MoveL Offs(p0,327.8320000000001,375.1264000000001, 0), v100, z5, tool0;
	MoveL Offs(p0,333.52,379.8046, 0), v100, z5, tool0;
	MoveL Offs(p0,339.352,384.15520000000004, 0), v100, z5, tool0;
	MoveL Offs(p0,345.4,388.225, 0), v100, z5, tool0;
	MoveL Offs(p0,351.736,392.06080000000003, 0), v100, z5, tool0;
	MoveL Offs(p0,358.43199999999996,395.7094, 0), v100, z5, tool0;
	MoveL Offs(p0,365.56000000000006,399.21760000000006, 0), v100, z5, tool0;
	MoveL Offs(p0,373.192,402.6322, 0), v100, z5, tool0;
	MoveL Offs(p0,381.4,406.0, 0), v100, z5, tool0;
	MoveL Offs(p0,389.7768000000001,409.2388, 0), v100, z5, tool0;
	MoveL Offs(p0,396.8864000000001,411.89440000000013, 0), v100, z5, tool0;
	MoveL Offs(p0,402.8776,413.9956, 0), v100, z5, tool0;
	MoveL Offs(p0,407.8992,415.57120000000003, 0), v100, z5, tool0;
	MoveL Offs(p0,412.1,416.65, 0), v100, z5, tool0;
	MoveL Offs(p0,415.62880000000007,417.2608, 0), v100, z5, tool0;
	MoveL Offs(p0,418.6344,417.43240000000003, 0), v100, z5, tool0;
	MoveL Offs(p0,421.2656,417.19359999999995, 0), v100, z5, tool0;
	MoveL Offs(p0,423.67120000000006,416.5732, 0), v100, z5, tool0;
	MoveL Offs(p0,426.0,415.6, 0), v100, z5, tool0;
	MoveL Offs(p0,429.1296000000001,414.26240000000007, 0), v100, z5, tool0;
	MoveL Offs(p0,430.57739999999995,413.8576, 0), v100, z5, tool0;
	MoveL Offs(p0,432.0768,413.6352, 0), v100, z5, tool0;
	MoveL Offs(p0,433.725,413.6, 0), v100, z5, tool0;
	MoveL Offs(p0,435.6192,413.75679999999994, 0), v100, z5, tool0;
	MoveL Offs(p0,437.85659999999996,414.1104, 0), v100, z5, tool0;
	MoveL Offs(p0,440.5344000000001,414.6656, 0), v100, z5, tool0;
	MoveL Offs(p0,443.74980000000005,415.42719999999997, 0), v100, z5, tool0;
	MoveL Offs(p0,447.6,416.4, 0), v100, z5, tool0;
	MoveL Offs(p0,452.6692000000001,417.53380000000004, 0), v100, z5, tool0;
	MoveL Offs(p0,457.8656000000001,418.4144000000001, 0), v100, z5, tool0;
	MoveL Offs(p0,463.1124,419.0406, 0), v100, z5, tool0;
	MoveL Offs(p0,468.33280000000013,419.4112000000001, 0), v100, z5, tool0;
	MoveL Offs(p0,473.45,419.525, 0), v100, z5, tool0;
	MoveL Offs(p0,478.3872,419.3808, 0), v100, z5, tool0;
	MoveL Offs(p0,483.0676,418.97739999999993, 0), v100, z5, tool0;
	MoveL Offs(p0,487.4144,418.31360000000006, 0), v100, z5, tool0;
	MoveL Offs(p0,491.3508,417.38820000000004, 0), v100, z5, tool0;
	MoveL Offs(p0,494.8,416.2, 0), v100, z5, tool0;
	MoveL Offs(p0,500.6,413.8, 0), v100, z5, tool0;
	MoveL Offs(p0,491.0,407.6, 0), v100, z5, tool0;
	MoveL Offs(p0,486.2446000000001,403.9768000000001, 0), v100, z5, tool0;
	MoveL Offs(p0,481.03680000000014,399.18240000000014, 0), v100, z5, tool0;
	MoveL Offs(p0,475.4642,393.3295999999999, 0), v100, z5, tool0;
	MoveL Offs(p0,469.61440000000005,386.53120000000007, 0), v100, z5, tool0;
	MoveL Offs(p0,463.575,378.9, 0), v100, z5, tool0;
	MoveL Offs(p0,457.43359999999996,370.5488, 0), v100, z5, tool0;
	MoveL Offs(p0,451.2778,361.5904, 0), v100, z5, tool0;
	MoveL Offs(p0,445.1952000000001,352.1376, 0), v100, z5, tool0;
	MoveL Offs(p0,439.27340000000004,342.3032, 0), v100, z5, tool0;
	MoveL Offs(p0,433.6,332.2, 0), v100, z5, tool0;
	MoveL Offs(p0,432.3858,330.0676, 0), v100, z5, tool0;
	MoveL Offs(p0,431.2544000000001,328.22080000000017, 0), v100, z5, tool0;
	MoveL Offs(p0,430.1926,326.6452, 0), v100, z5, tool0;
	MoveL Offs(p0,429.1872,325.32640000000004, 0), v100, z5, tool0;
	MoveL Offs(p0,428.225,324.25, 0), v100, z5, tool0;
	MoveL Offs(p0,427.2928,323.40160000000003, 0), v100, z5, tool0;
	MoveL Offs(p0,426.37739999999997,322.7668, 0), v100, z5, tool0;
	MoveL Offs(p0,425.4656,322.33119999999997, 0), v100, z5, tool0;
	MoveL Offs(p0,424.5442,322.0804, 0), v100, z5, tool0;
	MoveL Offs(p0,423.6,322.0, 0), v100, z5, tool0;
	MoveL Offs(p0,421.3656000000001,322.2092, 0), v100, z5, tool0;
	MoveL Offs(p0,419.0208000000001,322.8096000000001, 0), v100, z5, tool0;
	MoveL Offs(p0,416.6232,323.7604, 0), v100, z5, tool0;
	MoveL Offs(p0,414.23040000000003,325.0208, 0), v100, z5, tool0;
	MoveL Offs(p0,411.9,326.55, 0), v100, z5, tool0;
	MoveL Offs(p0,409.6896,328.3072, 0), v100, z5, tool0;
	MoveL Offs(p0,407.65680000000003,330.25159999999994, 0), v100, z5, tool0;
	MoveL Offs(p0,405.85920000000004,332.3424, 0), v100, z5, tool0;
	MoveL Offs(p0,404.35440000000006,334.53880000000004, 0), v100, z5, tool0;
	MoveL Offs(p0,403.2,336.8, 0), v100, z5, tool0;
	MoveL Offs(p0,400.7632000000001,341.206, 0), v100, z5, tool0;
	MoveL Offs(p0,397.3856000000001,345.26400000000007, 0), v100, z5, tool0;
	MoveL Offs(p0,393.2064,348.914, 0), v100, z5, tool0;
	MoveL Offs(p0,388.36480000000006,352.096, 0), v100, z5, tool0;
	MoveL Offs(p0,383.0,354.75, 0), v100, z5, tool0;
	MoveL Offs(p0,377.2512,356.816, 0), v100, z5, tool0;
	MoveL Offs(p0,371.2576,358.23400000000004, 0), v100, z5, tool0;
	MoveL Offs(p0,365.15840000000003,358.9440000000001, 0), v100, z5, tool0;
	MoveL Offs(p0,359.0928,358.88599999999997, 0), v100, z5, tool0;
	MoveL Offs(p0,353.2,358.0, 0), v100, z5, tool0;
	MoveL Offs(p0,349.63360000000006,357.1286, 0), v100, z5, tool0;
	MoveL Offs(p0,346.3168000000001,356.1648000000001, 0), v100, z5, tool0;
	MoveL Offs(p0,343.16319999999996,355.06419999999997, 0), v100, z5, tool0;
	MoveL Offs(p0,340.0864,353.78240000000005, 0), v100, z5, tool0;
	MoveL Offs(p0,337.0,352.275, 0), v100, z5, tool0;
	MoveL Offs(p0,333.8176,350.49760000000003, 0), v100, z5, tool0;
	MoveL Offs(p0,330.4528,348.4058, 0), v100, z5, tool0;
	MoveL Offs(p0,326.8192,345.95520000000005, 0), v100, z5, tool0;
	MoveL Offs(p0,322.8304,343.1014, 0), v100, z5, tool0;
	MoveL Offs(p0,318.4,339.8, 0), v100, z5, tool0;
	MoveL Offs(p0,313.32180000000005,336.14680000000004, 0), v100, z5, tool0;
	MoveL Offs(p0,308.7344000000001,333.3504000000001, 0), v100, z5, tool0;
	MoveL Offs(p0,304.5886,331.4155999999999, 0), v100, z5, tool0;
	MoveL Offs(p0,300.83520000000004,330.34720000000004, 0), v100, z5, tool0;
	MoveL Offs(p0,297.425,330.15, 0), v100, z5, tool0;
	MoveL Offs(p0,294.3088,330.8288, 0), v100, z5, tool0;
	MoveL Offs(p0,291.43739999999997,332.3884, 0), v100, z5, tool0;
	MoveL Offs(p0,288.7616,334.83360000000005, 0), v100, z5, tool0;
	MoveL Offs(p0,286.23220000000003,338.16920000000005, 0), v100, z5, tool0;
	MoveL Offs(p0,283.8,342.4, 0), v100, z5, tool0;
	MoveL Offs(p0,281.755,345.89660000000003, 0), v100, z5, tool0;
	MoveL Offs(p0,279.1520000000001,349.61280000000016, 0), v100, z5, tool0;
	MoveL Offs(p0,276.06899999999996,353.4682, 0), v100, z5, tool0;
	MoveL Offs(p0,272.584,357.3824, 0), v100, z5, tool0;
	MoveL Offs(p0,268.775,361.275, 0), v100, z5, tool0;
	MoveL Offs(p0,264.72,365.0656, 0), v100, z5, tool0;
	MoveL Offs(p0,260.497,368.6738, 0), v100, z5, tool0;
	MoveL Offs(p0,256.184,372.0192, 0), v100, z5, tool0;
	MoveL Offs(p0,251.859,375.02139999999997, 0), v100, z5, tool0;
	MoveL Offs(p0,247.6,377.6, 0), v100, z5, tool0;
	MoveL Offs(p0,243.5866,379.80140000000006, 0), v100, z5, tool0;
	MoveL Offs(p0,239.30080000000007,381.93920000000014, 0), v100, z5, tool0;
	MoveL Offs(p0,234.8542,383.9738, 0), v100, z5, tool0;
	MoveL Offs(p0,230.3584,385.86560000000003, 0), v100, z5, tool0;
	MoveL Offs(p0,225.925,387.575, 0), v100, z5, tool0;
	MoveL Offs(p0,221.66559999999998,389.06239999999997, 0), v100, z5, tool0;
	MoveL Offs(p0,217.6918,390.2882, 0), v100, z5, tool0;
	MoveL Offs(p0,214.11520000000002,391.2128, 0), v100, z5, tool0;
	MoveL Offs(p0,211.0474,391.7966, 0), v100, z5, tool0;
	MoveL Offs(p0,208.6,392.0, 0), v100, z5, tool0;
	MoveL Offs(p0,206.31080000000003,392.1102, 0), v100, z5, tool0;
	MoveL Offs(p0,204.85440000000008,392.4496000000001, 0), v100, z5, tool0;
	MoveL Offs(p0,204.2476,393.03139999999996, 0), v100, z5, tool0;
	MoveL Offs(p0,204.5072,393.8688, 0), v100, z5, tool0;
	MoveL Offs(p0,205.65,394.975, 0), v100, z5, tool0;
	MoveL Offs(p0,207.69279999999998,396.36319999999995, 0), v100, z5, tool0;
	MoveL Offs(p0,210.6524,398.0466, 0), v100, z5, tool0;
	MoveL Offs(p0,214.5456,400.0384, 0), v100, z5, tool0;
	MoveL Offs(p0,219.38920000000002,402.3518, 0), v100, z5, tool0;
	MoveL Offs(p0,225.2,405.0, 0), v100, z5, tool0;
	MoveL Offs(p0,242.01680000000002,412.23160000000007, 0), v100, z5, tool0;
	MoveL Offs(p0,259.1024000000001,419.12480000000016, 0), v100, z5, tool0;
	MoveL Offs(p0,276.26959999999997,425.6172, 0), v100, z5, tool0;
	MoveL Offs(p0,293.3312,431.6464000000001, 0), v100, z5, tool0;
	MoveL Offs(p0,310.1,437.15, 0), v100, z5, tool0;
	MoveL Offs(p0,326.3888,442.0656, 0), v100, z5, tool0;
	MoveL Offs(p0,342.0104,446.3308, 0), v100, z5, tool0;
	MoveL Offs(p0,356.7776,449.88320000000004, 0), v100, z5, tool0;
	MoveL Offs(p0,370.5032,452.66040000000004, 0), v100, z5, tool0;
	MoveL Offs(p0,383.0,454.6, 0), v100, z5, tool0;
	MoveL Offs(p0,386.4298,454.9782, 0), v100, z5, tool0;
	MoveL Offs(p0,390.4704000000001,455.27360000000016, 0), v100, z5, tool0;
	MoveL Offs(p0,394.9285999999999,455.4874, 0), v100, z5, tool0;
	MoveL Offs(p0,399.61120000000005,455.62080000000003, 0), v100, z5, tool0;
	MoveL Offs(p0,404.325,455.675, 0), v100, z5, tool0;
	MoveL Offs(p0,408.8768,455.65119999999996, 0), v100, z5, tool0;
	MoveL Offs(p0,413.07340000000005,455.5505999999999, 0), v100, z5, tool0;
	MoveL Offs(p0,416.7216,455.37440000000004, 0), v100, z5, tool0;
	MoveL Offs(p0,419.6282,455.1238, 0), v100, z5, tool0;
	MoveL Offs(p0,421.6,454.8, 0), v100, z5, tool0;
	MoveL Offs(p0,421.6,454.8, 0), v100, z5, tool0;
	MoveJ Offs(p0,52.0,415.0, 10), v100, z1, tool0;
	MoveL Offs(p0,51.25820000000001,412.91100000000006, 0), v100, z5, tool0;
	MoveL Offs(p0,50.481600000000014,410.86400000000015, 0), v100, z5, tool0;
	MoveL Offs(p0,49.6834,408.88899999999995, 0), v100, z5, tool0;
	MoveL Offs(p0,48.876799999999996,407.016, 0), v100, z5, tool0;
	MoveL Offs(p0,48.075,405.275, 0), v100, z5, tool0;
	MoveL Offs(p0,47.291199999999996,403.696, 0), v100, z5, tool0;
	MoveL Offs(p0,46.538599999999995,402.309, 0), v100, z5, tool0;
	MoveL Offs(p0,45.83040000000001,401.14400000000006, 0), v100, z5, tool0;
	MoveL Offs(p0,45.1798,400.231, 0), v100, z5, tool0;
	MoveL Offs(p0,44.6,399.6, 0), v100, z5, tool0;
	MoveL Offs(p0,42.32800000000001,398.576, 0), v100, z5, tool0;
	MoveL Offs(p0,42.075,399.025, 0), v100, z5, tool0;
	MoveL Offs(p0,41.936,399.816, 0), v100, z5, tool0;
	MoveL Offs(p0,41.904999999999994,400.979, 0), v100, z5, tool0;
	MoveL Offs(p0,41.976,402.54400000000004, 0), v100, z5, tool0;
	MoveL Offs(p0,42.14300000000001,404.541, 0), v100, z5, tool0;
	MoveL Offs(p0,42.4,407.0, 0), v100, z5, tool0;
	MoveL Offs(p0,42.95200000000001,410.82400000000007, 0), v100, z5, tool0;
	MoveL Offs(p0,43.434999999999995,413.012, 0), v100, z5, tool0;
	MoveL Offs(p0,44.032000000000004,415.32000000000005, 0), v100, z5, tool0;
	MoveL Offs(p0,44.725,417.7, 0), v100, z5, tool0;
	MoveL Offs(p0,45.496,420.104, 0), v100, z5, tool0;
	MoveL Offs(p0,46.327000000000005,422.48400000000004, 0), v100, z5, tool0;
	MoveL Offs(p0,47.2,424.79200000000003, 0), v100, z5, tool0;
	MoveL Offs(p0,48.097,426.98, 0), v100, z5, tool0;
	MoveL Offs(p0,49.0,429.0, 0), v100, z5, tool0;
	MoveL Offs(p0,50.5726,432.2454000000001, 0), v100, z5, tool0;
	MoveL Offs(p0,51.83680000000002,434.8032000000001, 0), v100, z5, tool0;
	MoveL Offs(p0,52.8322,436.7058, 0), v100, z5, tool0;
	MoveL Offs(p0,53.598400000000005,437.9856, 0), v100, z5, tool0;
	MoveL Offs(p0,54.175,438.675, 0), v100, z5, tool0;
	MoveL Offs(p0,54.601600000000005,438.80639999999994, 0), v100, z5, tool0;
	MoveL Offs(p0,54.9178,438.41220000000004, 0), v100, z5, tool0;
	MoveL Offs(p0,55.1632,437.5248, 0), v100, z5, tool0;
	MoveL Offs(p0,55.37740000000001,436.17659999999995, 0), v100, z5, tool0;
	MoveL Offs(p0,55.6,434.4, 0), v100, z5, tool0;
	MoveL Offs(p0,55.609600000000015,431.67200000000014, 0), v100, z5, tool0;
	MoveL Offs(p0,55.45239999999999,429.945, 0), v100, z5, tool0;
	MoveL Offs(p0,55.19680000000001,428.03200000000004, 0), v100, z5, tool0;
	MoveL Offs(p0,54.85,425.975, 0), v100, z5, tool0;
	MoveL Offs(p0,54.419200000000004,423.816, 0), v100, z5, tool0;
	MoveL Offs(p0,53.9116,421.5969999999999, 0), v100, z5, tool0;
	MoveL Offs(p0,53.3344,419.36, 0), v100, z5, tool0;
	MoveL Offs(p0,52.6948,417.14700000000005, 0), v100, z5, tool0;
	MoveL Offs(p0,52.0,415.0, 0), v100, z5, tool0;
	MoveL Offs(p0,52.0,415.0, 0), v100, z5, tool0;
	MoveJ Offs(p0,502.0,405.6, 10), v100, z1, tool0;
	MoveL Offs(p0,501.2256000000001,402.7408000000001, 0), v100, z5, tool0;
	MoveL Offs(p0,500.3313999999999,400.73819999999995, 0), v100, z5, tool0;
	MoveL Offs(p0,499.1648,398.4704, 0), v100, z5, tool0;
	MoveL Offs(p0,497.775,396.025, 0), v100, z5, tool0;
	MoveL Offs(p0,496.2112,393.4896, 0), v100, z5, tool0;
	MoveL Offs(p0,494.52259999999995,390.9518, 0), v100, z5, tool0;
	MoveL Offs(p0,492.75840000000005,388.49920000000003, 0), v100, z5, tool0;
	MoveL Offs(p0,490.9678,386.2194, 0), v100, z5, tool0;
	MoveL Offs(p0,489.2,384.2, 0), v100, z5, tool0;
	MoveL Offs(p0,484.4960000000002,379.9168000000001, 0), v100, z5, tool0;
	MoveL Offs(p0,481.12699999999995,377.3132, 0), v100, z5, tool0;
	MoveL Offs(p0,477.392,374.6064, 0), v100, z5, tool0;
	MoveL Offs(p0,473.525,371.95, 0), v100, z5, tool0;
	MoveL Offs(p0,469.76000000000005,369.49760000000003, 0), v100, z5, tool0;
	MoveL Offs(p0,466.33099999999996,367.4028, 0), v100, z5, tool0;
	MoveL Offs(p0,463.47200000000004,365.8192, 0), v100, z5, tool0;
	MoveL Offs(p0,461.41700000000003,364.9004, 0), v100, z5, tool0;
	MoveL Offs(p0,460.4,364.8, 0), v100, z5, tool0;
	MoveL Offs(p0,461.65440000000007,367.95040000000006, 0), v100, z5, tool0;
	MoveL Offs(p0,463.6166,370.87859999999995, 0), v100, z5, tool0;
	MoveL Offs(p0,466.2592000000001,374.45120000000003, 0), v100, z5, tool0;
	MoveL Offs(p0,469.425,378.475, 0), v100, z5, tool0;
	MoveL Offs(p0,472.95680000000004,382.7568, 0), v100, z5, tool0;
	MoveL Offs(p0,476.6974,387.1034, 0), v100, z5, tool0;
	MoveL Offs(p0,480.48960000000005,391.32160000000005, 0), v100, z5, tool0;
	MoveL Offs(p0,484.1762,395.2182, 0), v100, z5, tool0;
	MoveL Offs(p0,487.6,398.6, 0), v100, z5, tool0;
	MoveL Offs(p0,490.5304000000001,401.199, 0), v100, z5, tool0;
	MoveL Offs(p0,493.09120000000013,403.36000000000007, 0), v100, z5, tool0;
	MoveL Offs(p0,495.29679999999996,405.089, 0), v100, z5, tool0;
	MoveL Offs(p0,497.1616,406.392, 0), v100, z5, tool0;
	MoveL Offs(p0,498.7,407.275, 0), v100, z5, tool0;
	MoveL Offs(p0,499.9264,407.744, 0), v100, z5, tool0;
	MoveL Offs(p0,500.85519999999997,407.805, 0), v100, z5, tool0;
	MoveL Offs(p0,501.5008000000001,407.46400000000006, 0), v100, z5, tool0;
	MoveL Offs(p0,501.8776,406.72700000000003, 0), v100, z5, tool0;
	MoveL Offs(p0,502.0,405.6, 0), v100, z5, tool0;
	MoveL Offs(p0,502.0,405.6, 0), v100, z5, tool0;
	MoveJ Offs(p0,515.0,404.4, 10), v100, z1, tool0;
	MoveL Offs(p0,512.6815999999999,404.7668, 0), v100, z5, tool0;
	MoveL Offs(p0,512.2544,405.05920000000003, 0), v100, z5, tool0;
	MoveL Offs(p0,511.82480000000004,405.4044, 0), v100, z5, tool0;
	MoveL Offs(p0,511.4,405.8, 0), v100, z5, tool0;
	MoveL Offs(p0,514.775,405.6, 0), v100, z5, tool0;
	MoveL Offs(p0,514.9903999999999,405.33119999999997, 0), v100, z5, tool0;
	MoveL Offs(p0,515.1242,405.0696, 0), v100, z5, tool0;
	MoveL Offs(p0,515.1728,404.8224000000001, 0), v100, z5, tool0;
	MoveL Offs(p0,515.1326,404.59680000000003, 0), v100, z5, tool0;
	MoveL Offs(p0,515.0,404.4, 0), v100, z5, tool0;
	MoveL Offs(p0,515.0,404.4, 0), v100, z5, tool0;
	MoveJ Offs(p0,524.8,397.6, 10), v100, z1, tool0;
	MoveL Offs(p0,526.1424000000001,395.5712000000001, 0), v100, z5, tool0;
	MoveL Offs(p0,526.5586,394.79380000000003, 0), v100, z5, tool0;
	MoveL Offs(p0,526.8032000000001,394.1376, 0), v100, z5, tool0;
	MoveL Offs(p0,526.875,393.575, 0), v100, z5, tool0;
	MoveL Offs(p0,526.7728,393.0784, 0), v100, z5, tool0;
	MoveL Offs(p0,526.4954,392.62019999999995, 0), v100, z5, tool0;
	MoveL Offs(p0,526.0416000000001,392.1728, 0), v100, z5, tool0;
	MoveL Offs(p0,525.4102,391.70860000000005, 0), v100, z5, tool0;
	MoveL Offs(p0,524.6,391.2, 0), v100, z5, tool0;
	MoveL Offs(p0,518.2706000000001,386.36800000000005, 0), v100, z5, tool0;
	MoveL Offs(p0,513.3248000000001,379.9040000000001, 0), v100, z5, tool0;
	MoveL Offs(p0,509.7661999999999,372.156, 0), v100, z5, tool0;
	MoveL Offs(p0,507.59839999999997,363.4720000000001, 0), v100, z5, tool0;
	MoveL Offs(p0,506.825,354.2, 0), v100, z5, tool0;
	MoveL Offs(p0,507.44960000000003,344.688, 0), v100, z5, tool0;
	MoveL Offs(p0,509.4758,335.284, 0), v100, z5, tool0;
	MoveL Offs(p0,512.9072,326.33600000000007, 0), v100, z5, tool0;
	MoveL Offs(p0,517.7474,318.192, 0), v100, z5, tool0;
	MoveL Offs(p0,524.0,311.2, 0), v100, z5, tool0;
	MoveL Offs(p0,526.3584000000002,308.9664000000001, 0), v100, z5, tool0;
	MoveL Offs(p0,527.3965999999999,307.9096, 0), v100, z5, tool0;
	MoveL Offs(p0,528.3232,306.9152, 0), v100, z5, tool0;
	MoveL Offs(p0,529.125,306.0, 0), v100, z5, tool0;
	MoveL Offs(p0,529.7888,305.1808, 0), v100, z5, tool0;
	MoveL Offs(p0,530.3014000000001,304.4744, 0), v100, z5, tool0;
	MoveL Offs(p0,530.6496000000001,303.89760000000007, 0), v100, z5, tool0;
	MoveL Offs(p0,530.8202,303.46720000000005, 0), v100, z5, tool0;
	MoveL Offs(p0,530.8,303.2, 0), v100, z5, tool0;
	MoveL Offs(p0,533.7340000000002,302.78520000000003, 0), v100, z5, tool0;
	MoveL Offs(p0,538.0800000000002,300.34560000000005, 0), v100, z5, tool0;
	MoveL Offs(p0,543.854,296.0484, 0), v100, z5, tool0;
	MoveL Offs(p0,550.672,290.2608, 0), v100, z5, tool0;
	MoveL Offs(p0,558.15,283.35, 0), v100, z5, tool0;
	MoveL Offs(p0,565.9040000000001,275.68319999999994, 0), v100, z5, tool0;
	MoveL Offs(p0,573.55,267.6276, 0), v100, z5, tool0;
	MoveL Offs(p0,580.7040000000001,259.55039999999997, 0), v100, z5, tool0;
	MoveL Offs(p0,586.982,251.8188, 0), v100, z5, tool0;
	MoveL Offs(p0,592.0,244.8, 0), v100, z5, tool0;
	MoveL Offs(p0,596.5132,237.4056, 0), v100, z5, tool0;
	MoveL Offs(p0,600.6736000000002,229.56480000000005, 0), v100, z5, tool0;
	MoveL Offs(p0,604.4523999999999,221.3712, 0), v100, z5, tool0;
	MoveL Offs(p0,607.8208000000001,212.91840000000002, 0), v100, z5, tool0;
	MoveL Offs(p0,610.75,204.3, 0), v100, z5, tool0;
	MoveL Offs(p0,613.2112,195.6096, 0), v100, z5, tool0;
	MoveL Offs(p0,615.1755999999999,186.9408, 0), v100, z5, tool0;
	MoveL Offs(p0,616.6144,178.3872, 0), v100, z5, tool0;
	MoveL Offs(p0,617.4988000000001,170.0424, 0), v100, z5, tool0;
	MoveL Offs(p0,617.8,162.0, 0), v100, z5, tool0;
	MoveL Offs(p0,617.6954000000001,157.42880000000002, 0), v100, z5, tool0;
	MoveL Offs(p0,617.2752000000002,152.52640000000002, 0), v100, z5, tool0;
	MoveL Offs(p0,616.5598,147.36960000000002, 0), v100, z5, tool0;
	MoveL Offs(p0,615.5696,142.0352, 0), v100, z5, tool0;
	MoveL Offs(p0,614.325,136.6, 0), v100, z5, tool0;
	MoveL Offs(p0,612.8464,131.14079999999998, 0), v100, z5, tool0;
	MoveL Offs(p0,611.1542,125.73440000000001, 0), v100, z5, tool0;
	MoveL Offs(p0,609.2688,120.4576, 0), v100, z5, tool0;
	MoveL Offs(p0,607.2106,115.3872, 0), v100, z5, tool0;
	MoveL Offs(p0,605.0,110.6, 0), v100, z5, tool0;
	MoveL Offs(p0,600.0554000000001,101.97680000000001, 0), v100, z5, tool0;
	MoveL Offs(p0,594.0992000000002,94.05440000000004, 0), v100, z5, tool0;
	MoveL Offs(p0,587.3078,86.93359999999998, 0), v100, z5, tool0;
	MoveL Offs(p0,579.8576,80.71520000000001, 0), v100, z5, tool0;
	MoveL Offs(p0,571.925,75.5, 0), v100, z5, tool0;
	MoveL Offs(p0,563.6864,71.38879999999999, 0), v100, z5, tool0;
	MoveL Offs(p0,555.3181999999999,68.4824, 0), v100, z5, tool0;
	MoveL Offs(p0,546.9968000000001,66.8816, 0), v100, z5, tool0;
	MoveL Offs(p0,538.8986,66.6872, 0), v100, z5, tool0;
	MoveL Offs(p0,531.2,68.0, 0), v100, z5, tool0;
	MoveL Offs(p0,527.2374,69.34020000000001, 0), v100, z5, tool0;
	MoveL Offs(p0,523.5232000000002,71.06560000000002, 0), v100, z5, tool0;
	MoveL Offs(p0,520.0778,73.15339999999999, 0), v100, z5, tool0;
	MoveL Offs(p0,516.9216,75.58080000000001, 0), v100, z5, tool0;
	MoveL Offs(p0,514.075,78.325, 0), v100, z5, tool0;
	MoveL Offs(p0,511.5584,81.3632, 0), v100, z5, tool0;
	MoveL Offs(p0,509.39219999999995,84.6726, 0), v100, z5, tool0;
	MoveL Offs(p0,507.5968000000001,88.2304, 0), v100, z5, tool0;
	MoveL Offs(p0,506.19259999999997,92.01380000000002, 0), v100, z5, tool0;
	MoveL Offs(p0,505.2,96.0, 0), v100, z5, tool0;
	MoveL Offs(p0,504.73600000000016,99.1568, 0), v100, z5, tool0;
	MoveL Offs(p0,504.62399999999997,100.12019999999998, 0), v100, z5, tool0;
	MoveL Offs(p0,504.60800000000006,100.6624, 0), v100, z5, tool0;
	MoveL Offs(p0,504.7,100.775, 0), v100, z5, tool0;
	MoveL Offs(p0,504.912,100.4496, 0), v100, z5, tool0;
	MoveL Offs(p0,505.256,99.6778, 0), v100, z5, tool0;
	MoveL Offs(p0,505.744,98.4512, 0), v100, z5, tool0;
	MoveL Offs(p0,507.2,94.6, 0), v100, z5, tool0;
	MoveL Offs(p0,508.3916000000001,91.93340000000002, 0), v100, z5, tool0;
	MoveL Offs(p0,509.9888000000001,89.15520000000002, 0), v100, z5, tool0;
	MoveL Offs(p0,511.9052,86.35779999999998, 0), v100, z5, tool0;
	MoveL Offs(p0,514.0544000000001,83.6336, 0), v100, z5, tool0;
	MoveL Offs(p0,516.35,81.075, 0), v100, z5, tool0;
	MoveL Offs(p0,518.7056,78.77439999999999, 0), v100, z5, tool0;
	MoveL Offs(p0,521.0348,76.82419999999999, 0), v100, z5, tool0;
	MoveL Offs(p0,523.2512,75.31680000000001, 0), v100, z5, tool0;
	MoveL Offs(p0,525.2684,74.3446, 0), v100, z5, tool0;
	MoveL Offs(p0,527.0,74.0, 0), v100, z5, tool0;
	MoveL Offs(p0,529.1,73.5, 0), v100, z5, tool0;
	MoveL Offs(p0,529.4048,73.30879999999999, 0), v100, z5, tool0;
	MoveL Offs(p0,529.6544,73.0984, 0), v100, z5, tool0;
	MoveL Offs(p0,529.8416000000001,72.87360000000001, 0), v100, z5, tool0;
	MoveL Offs(p0,529.9592,72.6392, 0), v100, z5, tool0;
	MoveL Offs(p0,530.0,72.4, 0), v100, z5, tool0;
	MoveL Offs(p0,532.4576000000001,71.38080000000001, 0), v100, z5, tool0;
	MoveL Offs(p0,535.2164,71.4802, 0), v100, z5, tool0;
	MoveL Offs(p0,538.7167999999999,71.9264, 0), v100, z5, tool0;
	MoveL Offs(p0,542.75,72.675, 0), v100, z5, tool0;
	MoveL Offs(p0,547.1072,73.6816, 0), v100, z5, tool0;
	MoveL Offs(p0,551.5795999999999,74.90180000000001, 0), v100, z5, tool0;
